KUKA KRL program: MyProgram_245().src

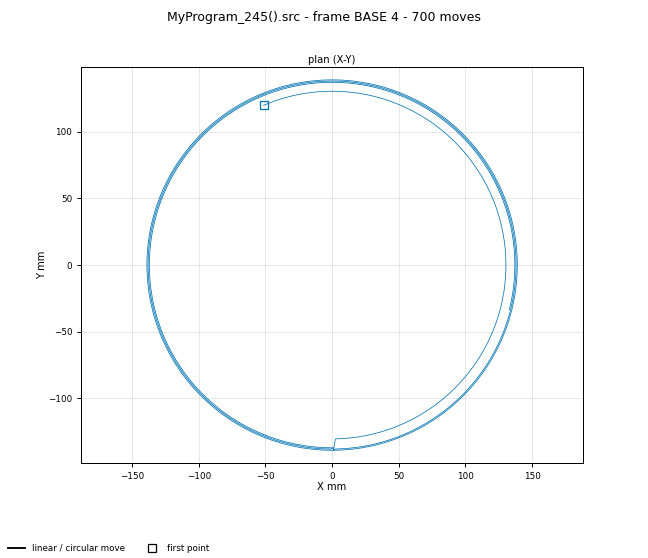
[picture p0: tool path of MyProgram_245().src in frame BASE 4, 700 of 700 moves have a stored position in this frame; points joined in program order, loops and branches not executed]
&ACCESS RVP
&REL 1
&PARAM TEMPLATE = C:\KRC\Roboter\Template\vorgabe
&PARAM EDITMASK = *
DEF MyProgram_245()
; ---- Setting reference (Base) ----
$BASE = BASE_DATA[4]

; --------------------------
; ---- Setting tool (TCP) ----
$TOOL = TOOL_DATA[3]
; --------------------------

$VEL.CP = VEL_APROX_PRINT
Startdeposition()
$VEL.CP = VEL_PRINT
LIN {X -51.3648,Y 119.8382,Z 162,A 112.229,B 13.3996,C -0.1433,E1 13.3387,E2 337.7554} C_DIS
LIN {X -48.41,Y 121.0619,Z 162,A 110.818,B 13.3996,C -0.1448,E1 13.3424,E2 339.1659} C_DIS
LIN {X -45.4271,Y 122.2124,Z 162,A 109.4036,B 13.3996,C -0.1461,E1 13.3461,E2 340.5802} C_DIS
LIN {X -41.7334,Y 123.5235,Z 162,A 107.6109,B 13.3996,C -0.1461,E1 13.3508,E2 342.3795} C_DIS
LIN {X -37.8366,Y 124.7715,Z 162,A 105.8754,B 13.3995,C -0.1495,E1 13.3554,E2 344.1065} C_DIS
LIN {X -34.901,Y 125.624,Z 162,A 104.5108,B 13.3995,C -0.1501,E1 13.3591,E2 345.4724} C_DIS
LIN {X -31.641,Y 126.4851,Z 162,A 102.9054,B 13.3995,C -0.1482,E1 13.3635,E2 347.0909} C_DIS
LIN {X -27.3855,Y 127.4735,Z 162,A 101.0691,B 13.3995,C -0.1517,E1 13.3684,E2 348.9163} C_DIS
LIN {X -23.8932,Y 128.1754,Z 162,A 99.5551,B 13.3995,C -0.154,E1 13.3726,E2 350.4234} C_DIS
LIN {X -20.7831,Y 128.7167,Z 162,A 98.1393,B 13.3995,C -0.154,E1 13.3765,E2 351.8415} C_DIS
LIN {X -17.5414,Y 129.1981,Z 162,A 96.6995,B 13.3995,C -0.1548,E1 13.3805,E2 353.2805} C_DIS
LIN {X -14.3691,Y 129.5885,Z 162,A 95.137,B 13.3995,C -0.1513,E1 13.3848,E2 354.8601} C_DIS
LIN {X -10.509,Y 129.9587,Z 162,A 93.576,B 13.3995,C -0.1556,E1 13.3891,E2 356.4038} C_DIS
LIN {X -6.3901,Y 130.2256,Z 162,A 91.7902,B 13.3995,C -0.1568,E1 13.3941,E2 358.1854} C_DIS
LIN {X -2.5144,Y 130.3584,Z 162,A 90.0176,B 13.3995,C -0.1553,E1 13.3991,E2 359.9649} C_DIS
LIN {X 0.6814,Y 130.3805,Z 162,A 88.6373,B 13.3995,C -0.156,E1 13.4029,E2 361.3419} C_DIS
LIN {X 4.7953,Y 130.2943,Z 162,A 86.8534,B 13.3995,C -0.1566,E1 13.4079,E2 363.1222} C_DIS
LIN {X 8.3824,Y 130.1129,Z 162,A 85.186,B 13.3995,C -0.1541,E1 13.4126,E2 364.7991} C_DIS
LIN {X 11.8671,Y 129.8423,Z 162,A 83.7187,B 13.3995,C -0.1557,E1 13.4166,E2 366.2581} C_DIS
LIN {X 15.283,Y 129.4833,Z 162,A 82.2394,B 13.3995,C -0.1561,E1 13.4207,E2 367.7333} C_DIS
LIN {X 18.2152,Y 129.1036,Z 162,A 80.8926,B 13.3995,C -0.1544,E1 13.4244,E2 369.0852} C_DIS
LIN {X 21.6827,Y 128.5666,Z 162,A 79.4104,B 13.3995,C -0.1554,E1 13.4285,E2 370.5601} C_DIS
LIN {X 24.8115,Y 127.9998,Z 162,A 78.0162,B 13.3995,C -0.1548,E1 13.4323,E2 371.9536} C_DIS
LIN {X 27.9273,Y 127.3565,Z 162,A 76.6207,B 13.3995,C -0.1541,E1 13.4362,E2 373.3485} C_DIS
LIN {X 31.6838,Y 126.4742,Z 162,A 74.7821,B 13.3995,C -0.1492,E1 13.4412,E2 375.2032} C_DIS
LIN {X 35.6775,Y 125.4068,Z 162,A 73.1149,B 13.3995,C -0.152,E1 13.4456,E2 376.853} C_DIS
LIN {X 39.3818,Y 124.2923,Z 162,A 71.2587,B 13.3995,C -0.1463,E1 13.4506,E2 378.727} C_DIS
LIN {X 43.2866,Y 122.988,Z 162,A 69.6267,B 13.3995,C -0.1496,E1 13.4549,E2 380.3385} C_DIS
LIN {X 46.2866,Y 121.8905,Z 162,A 68.2137,B 13.3995,C -0.148,E1 13.4586,E2 381.7524} C_DIS
LIN {X 49.8892,Y 120.4599,Z 162,A 66.4224,B 13.3995,C -0.1437,E1 13.4632,E2 383.5538} C_DIS
LIN {X 53.6946,Y 118.8129,Z 162,A 64.5724,B 13.3995,C -0.1409,E1 13.468,E2 385.4071} C_DIS
LIN {X 57.8056,Y 116.867,Z 162,A 62.6784,B 13.3995,C -0.1414,E1 13.4727,E2 387.2891} C_DIS
LIN {X 61.4635,Y 114.9879,Z 162,A 60.9224,B 13.3995,C -0.1405,E1 13.477,E2 389.0395} C_DIS
LIN {X 64.2616,Y 113.4482,Z 162,A 59.5277,B 13.3995,C -0.1388,E1 13.4804,E2 390.4334} C_DIS
LIN {X 67.0341,Y 111.8321,Z 162,A 57.9785,B 13.3997,C -0.1328,E1 13.4842,E2 391.999} C_DIS
LIN {X 70.5604,Y 109.6413,Z 162,A 56.3411,B 13.3997,C -0.1353,E1 13.488,E2 393.6151} C_DIS
LIN {X 73.2045,Y 107.8935,Z 162,A 54.9184,B 13.3997,C -0.1322,E1 13.4913,E2 395.0416} C_DIS
LIN {X 76.3807,Y 105.6688,Z 162,A 53.2322,B 13.3997,C -0.1299,E1 13.4952,E2 396.7262} C_DIS
LIN {X 79.5821,Y 103.2797,Z 162,A 51.4056,B 13.3997,C -0.1248,E1 13.4993,E2 398.5616} C_DIS
LIN {X 82.7084,Y 100.7932,Z 162,A 49.6058,B 13.3997,C -0.1204,E1 13.5032,E2 400.3672} C_DIS
LIN {X 86.1178,Y 97.8964,Z 162,A 47.6543,B 13.3997,C -0.1171,E1 13.5073,E2 402.3178} C_DIS
LIN {X 89.3226,Y 94.981,Z 162,A 45.8282,B 13.3998,C -0.1156,E1 13.511,E2 404.1357} C_DIS
LIN {X 92.196,Y 92.1952,Z 162,A 44.047,B 13.3998,C -0.1114,E1 13.5146,E2 405.9204} C_DIS
LIN {X 94.98,Y 89.3237,Z 162,A 42.3244,B 13.3998,C -0.1087,E1 13.5179,E2 407.6398} C_DIS
LIN {X 97.8953,Y 86.119,Z 162,A 40.4215,B 13.3999,C -0.1046,E1 13.5214,E2 409.5436} C_DIS
LIN {X 100.577,Y 82.9711,Z 162,A 38.6615,B 13.3999,C -0.1023,E1 13.5246,E2 411.298} C_DIS
LIN {X 103.0711,Y 79.8514,Z 162,A 36.9109,B 13.3999,C -0.0984,E1 13.5276,E2 413.0491} C_DIS
LIN {X 105.6784,Y 76.3675,Z 162,A 35.0847,B 13.3999,C -0.0964,E1 13.5306,E2 414.8666} C_DIS
LIN {X 107.8606,Y 73.2531,Z 162,A 33.3672,B 13.3999,C -0.091,E1 13.5334,E2 416.5905} C_DIS
LIN {X 109.7275,Y 70.4258,Z 162,A 31.8007,B 13.4,C -0.0851,E1 13.5358,E2 418.1672} C_DIS
LIN {X 112.0026,Y 66.748,Z 162,A 29.9637,B 13.4,C -0.0822,E1 13.5384,E2 419.9982} C_DIS
LIN {X 113.8971,Y 63.4622,Z 162,A 28.287,B 13.4,C -0.0777,E1 13.5407,E2 421.6773} C_DIS
LIN {X 116.0401,Y 59.4489,Z 162,A 26.3867,B 13.4,C -0.0754,E1 13.5432,E2 423.5676} C_DIS
LIN {X 117.5653,Y 56.3719,Z 162,A 24.978,B 13.4,C -0.0744,E1 13.5449,E2 424.9657} C_DIS
LIN {X 119.0932,Y 53.0681,Z 162,A 23.3299,B 13.4001,C -0.0687,E1 13.5468,E2 426.6209} C_DIS
LIN {X 120.4588,Y 49.8919,Z 162,A 21.8599,B 13.4001,C -0.0661,E1 13.5484,E2 428.0865} C_DIS
LIN {X 121.6461,Y 46.9227,Z 162,A 20.4706,B 13.4001,C -0.0627,E1 13.5498,E2 429.4752} C_DIS
LIN {X 122.9568,Y 43.3767,Z 162,A 18.7812,B 13.4001,C -0.0572,E1 13.5514,E2 431.1694} C_DIS
LIN {X 124.0954,Y 39.9981,Z 162,A 17.1481,B 13.4002,C -0.0509,E1 13.5529,E2 432.8117} C_DIS
LIN {X 125.2249,Y 36.308,Z 162,A 15.6024,B 13.4002,C -0.0506,E1 13.5541,E2 434.3415} C_DIS
LIN {X 126.0759,Y 33.2329,Z 162,A 14.2165,B 13.4002,C -0.0471,E1 13.5551,E2 435.7269} C_DIS
LIN {X 126.8513,Y 30.1389,Z 162,A 12.8316,B 13.4002,C -0.0435,E1 13.556,E2 437.1112} C_DIS
LIN {X 127.5503,Y 27.0298,Z 162,A 11.4491,B 13.4002,C -0.04,E1 13.5568,E2 438.4931} C_DIS
LIN {X 128.172,Y 23.9106,Z 162,A 10.0677,B 13.4002,C -0.0364,E1 13.5576,E2 439.874} C_DIS
LIN {X 128.7292,Y 20.7083,Z 162,A 8.6371,B 13.4002,C -0.0322,E1 13.5582,E2 441.3064} C_DIS
LIN {X 129.1974,Y 17.5462,Z 162,A 7.2474,B 13.4002,C -0.0285,E1 13.5588,E2 442.6959} C_DIS
LIN {X 129.588,Y 14.3743,Z 162,A 5.7046,B 13.4002,C -0.0202,E1 13.5593,E2 444.2564} C_DIS
LIN {X 129.9579,Y 10.5182,Z 162,A 4.1609,B 13.4002,C -0.0199,E1 13.5597,E2 445.7833} C_DIS
LIN {X 130.1912,Y 7.0747,Z 162,A 2.7517,B 13.4002,C -0.0187,E1 13.5599,E2 447.1816} C_DIS
LIN {X 130.3247,Y 3.8815,Z 162,A 1.1882,B 13.4002,C -0.0097,E1 13.5601,E2 448.7654} C_DIS
LIN {X 130.3848,Y 0.1344,Z 162,A -0.3942,B 13.4003,C -0.0067,E1 13.5601,E2 450.3422} C_DIS
LIN {X 130.3585,Y -2.5119,Z 162,A -1.618,B 13.4003,C -0.0014,E1 13.5601,E2 451.5745} C_DIS
LIN {X 130.2251,Y -6.3989,Z 162,A -3.2663,B 13.4003,C 0.0019,E1 13.5598,E2 453.2176} C_DIS
LIN {X 129.9591,Y -10.5042,Z 162,A -4.89,B 13.4003,C 0.0017,E1 13.5595,E2 454.8217} C_DIS
LIN {X 129.6619,Y -13.6875,Z 162,A -6.3508,B 13.4003,C 0.0076,E1 13.5591,E2 456.2907} C_DIS
LIN {X 129.2869,Y -16.8636,Z 162,A -7.6852,B 13.4003,C 0.0096,E1 13.5587,E2 457.6185} C_DIS
LIN {X 128.8327,Y -20.0401,Z 162,A -9.1175,B 13.4003,C 0.0145,E1 13.5581,E2 459.0551} C_DIS
LIN {X 128.2705,Y -23.3733,Z 162,A -10.5754,B 13.4003,C 0.018,E1 13.5574,E2 460.5116} C_DIS
LIN {X 127.6866,Y -26.3768,Z 162,A -11.922,B 13.4003,C 0.0221,E1 13.5566,E2 461.8601} C_DIS
LIN {X 127.0065,Y -29.4789,Z 162,A -13.3152,B 13.4003,C 0.0261,E1 13.5558,E2 463.2547} C_DIS
LIN {X 125.9936,Y -33.5417,Z 162,A -15.217,B 13.4003,C 0.0333,E1 13.5545,E2 465.1661} C_DIS
LIN {X 124.9621,Y -37.2055,Z 162,A -16.9347,B 13.4003,C 0.0396,E1 13.5531,E2 466.8912} C_DIS
LIN {X 123.5101,Y -41.7736,Z 162,A -18.8648,B 13.4003,C 0.0403,E1 13.5515,E2 468.8031} C_DIS
LIN {X 122.2133,Y -45.4248,Z 162,A -20.5475,B 13.4003,C 0.0445,E1 13.5499,E2 470.4855} C_DIS
LIN {X 120.7527,Y -49.1771,Z 162,A -22.324,B 13.4003,C 0.0497,E1 13.548,E2 472.2651} C_DIS
LIN {X 119.4381,Y -52.2904,Z 162,A -23.7684,B 13.4003,C 0.0526,E1 13.5464,E2 473.7065} C_DIS
LIN {X 117.86,Y -55.7553,Z 162,A -25.5751,B 13.4002,C 0.0613,E1 13.5443,E2 475.5311} C_DIS
LIN {X 116.0429,Y -59.4433,Z 162,A -27.3002,B 13.4002,C 0.0638,E1 13.5421,E2 477.2488} C_DIS
LIN {X 113.8942,Y -63.4675,Z 162,A -29.2997,B 13.4002,C 0.069,E1 13.5395,E2 479.2503} C_DIS
LIN {X 111.8352,Y -67.0289,Z 162,A -30.9899,B 13.4002,C 0.0702,E1 13.5371,E2 480.9287} C_DIS
LIN {X 109.7887,Y -70.3302,Z 162,A -32.6796,B 13.4002,C 0.0741,E1 13.5346,E2 482.6185} C_DIS
LIN {X 107.8875,Y -73.2133,Z 162,A -34.1796,B 13.4001,C 0.0775,E1 13.5323,E2 484.1183} C_DIS
LIN {X 105.67,Y -76.3791,Z 162,A -35.979,B 13.4001,C 0.0848,E1 13.5293,E2 485.9318} C_DIS
LIN {X 103.2272,Y -79.6499,Z 162,A -37.7816,B 13.4001,C 0.0894,E1 13.5263,E2 487.7375} C_DIS
LIN {X 100.5472,Y -83.0071,Z 162,A -39.5954,B 13.4,C 0.0918,E1 13.5231,E2 489.5448} C_DIS
LIN {X 97.8942,Y -86.1203,Z 162,A -41.3629,B 13.4,C 0.0951,E1 13.5199,E2 491.3109} C_DIS
LIN {X 95.1164,Y -89.1791,Z 162,A -43.2237,B 13.4,C 0.1006,E1 13.5163,E2 493.1792} C_DIS
LIN {X 92.1564,Y -92.2345,Z 162,A -45.0418,B 13.4,C 0.1032,E1 13.5128,E2 494.9933} C_DIS
LIN {X 89.3105,Y -94.9924,Z 162,A -46.7553,B 13.3999,C 0.1062,E1 13.5093,E2 496.7055} C_DIS
LIN {X 86.1673,Y -97.8526,Z 162,A -48.6377,B 13.3999,C 0.1105,E1 13.5054,E2 498.5918} C_DIS
LIN {X 82.9551,Y -100.5903,Z 162,A -50.4234,B 13.3999,C 0.1122,E1 13.5016,E2 500.3714} C_DIS
LIN {X 79.843,Y -103.0775,Z 162,A -52.1734,B 13.3999,C 0.1156,E1 13.4978,E2 502.1232} C_DIS
LIN {X 77.1216,Y -105.1292,Z 162,A -53.6275,B 13.3998,C 0.1172,E1 13.4945,E2 503.5738} C_DIS
LIN {X 73.7716,Y -107.5064,Z 162,A -55.3844,B 13.3998,C 0.1191,E1 13.4905,E2 505.3268} C_DIS
LIN {X 70.5219,Y -109.666,Z 162,A -57.1358,B 13.3998,C 0.1231,E1 13.4864,E2 507.0844} C_DIS
LIN {X 67.6092,Y -111.485,Z 162,A -58.5789,B 13.3998,C 0.1238,E1 13.483,E2 508.5212} C_DIS
LIN {X 64.8583,Y -113.1078,Z 162,A -59.9789,B 13.3998,C 0.1259,E1 13.4796,E2 509.9222} C_DIS
LIN {X 61.4575,Y -114.9911,Z 162,A -61.8495,B 13.3997,C 0.1333,E1 13.4749,E2 511.8137} C_DIS
LIN {X 57.8054,Y -116.8671,Z 162,A -63.582,B 13.3997,C 0.1339,E1 13.4706,E2 513.5393} C_DIS
LIN {X 54.3123,Y -118.5316,Z 162,A -65.1666,B 13.3997,C 0.1329,E1 13.4667,E2 515.1117} C_DIS
LIN {X 51.3578,Y -119.8413,Z 162,A -66.5759,B 13.3997,C 0.1345,E1 13.4631,E2 516.5211} C_DIS
LIN {X 48.4058,Y -121.0636,Z 162,A -67.9724,B 13.3997,C 0.136,E1 13.4594,E2 517.9179} C_DIS
LIN {X 45.4242,Y -122.2135,Z 162,A -69.3694,B 13.3997,C 0.1375,E1 13.4558,E2 519.3152} C_DIS
LIN {X 41.7737,Y -123.5101,Z 162,A -71.1872,B 13.3996,C 0.1427,E1 13.451,E2 521.1482} C_DIS
LIN {X 38.3453,Y -124.6158,Z 162,A -72.7502,B 13.3996,C 0.1437,E1 13.4468,E2 522.7101} C_DIS
LIN {X 34.7135,Y -125.6764,Z 162,A -74.2918,B 13.3996,C 0.1419,E1 13.4427,E2 524.2387} C_DIS
LIN {X 31.3975,Y -126.5469,Z 162,A -75.9774,B 13.3995,C 0.1483,E1 13.4381,E2 525.9467} C_DIS
LIN {X 26.998,Y -127.5572,Z 162,A -77.7693,B 13.3995,C 0.1444,E1 13.4332,E2 527.7173} C_DIS
LIN {X 23.9433,Y -128.1658,Z 162,A -79.1368,B 13.3995,C 0.1454,E1 13.4295,E2 529.0855} C_DIS
LIN {X 20.714,Y -128.7282,Z 162,A -80.5881,B 13.3995,C 0.1466,E1 13.4255,E2 530.5391} C_DIS
LIN {X 17.8284,Y -129.1588,Z 162,A -81.9277,B 13.3995,C 0.1489,E1 13.4218,E2 531.8863} C_DIS
LIN {X 14.3642,Y -129.5891,Z 162,A -83.5544,B 13.3995,C 0.1522,E1 13.4172,E2 533.5249} C_DIS
LIN {X 10.5051,Y -129.9591,Z 162,A -85.1137,B 13.3995,C 0.1489,E1 13.4129,E2 535.0681} C_DIS
LIN {X 6.3995,Y -130.2251,Z 162,A -86.8884,B 13.3995,C 0.1486,E1 13.408,E2 536.8399} C_DIS
LIN {X 2.5092,Y -130.3585,Z 162,A -88.632,B 13.3995,C 0.1499,E1 13.4031,E2 538.5883} C_DIS
LIN {X 2.5092,Y -130.3585,Z 162,A -88.632,B 13.3995,C 0.1499,E1 13.4031,E2 538.5883} C_DIS
Enddeposition()
LIN {X 0.9764,Y -138.8979,Z 163,A -92.574,B 24.9723,C -1.2156,E1 25.0012,E2 539.334} C_DIS
Startdeposition()
$VEL.CP = VEL_PRINT
LIN {X -2.6014,Y -138.8804,Z 163,A -94.2722,B 24.9729,C -1.203,E1 24.9963,E2 541.0621} C_DIS
LIN {X -5.7121,Y -138.7872,Z 163,A -95.5603,B 24.9729,C -1.2026,E1 24.9927,E2 542.3514} C_DIS
LIN {X -9.5587,Y -138.5762,Z 163,A -97.2235,B 24.9731,C -1.1985,E1 24.9881,E2 544.0249} C_DIS
LIN {X -13.6038,Y -138.2369,Z 163,A -98.8717,B 24.9731,C -1.2,E1 24.9835,E2 545.6702} C_DIS
LIN {X -17.9643,Y -137.7377,Z 163,A -100.6653,B 24.973,C -1.2013,E1 24.9785,E2 547.4622} C_DIS
LIN {X -21.6009,Y -137.2148,Z 163,A -102.1377,B 24.9729,C -1.204,E1 24.9745,E2 548.9293} C_DIS
LIN {X -25.0156,Y -136.6341,Z 163,A -103.5921,B 24.9729,C -1.2031,E1 24.9705,E2 550.3873} C_DIS
LIN {X -30.6353,Y -135.484,Z 163,A -105.7443,B 24.9723,C -1.2158,E1 24.9647,E2 552.5119} C_DIS
LIN {X -34.265,Y -134.6115,Z 163,A -107.5105,B 24.9728,C -1.2044,E1 24.9598,E2 554.3077} C_DIS
LIN {X -37.6332,Y -133.7091,Z 163,A -108.97,B 24.9728,C -1.2042,E1 24.9559,E2 555.7699} C_DIS
LIN {X -41.7719,Y -132.4752,Z 163,A -110.7909,B 24.9728,C -1.2034,E1 24.951,E2 557.5958} C_DIS
LIN {X -45.7264,Y -131.162,Z 163,A -112.4532,B 24.9727,C -1.2079,E1 24.9466,E2 559.2506} C_DIS
LIN {X -49.4255,Y -129.8152,Z 163,A -114.0534,B 24.9726,C -1.2107,E1 24.9424,E2 560.8475} C_DIS
LIN {X -52.632,Y -128.5486,Z 163,A -115.574,B 24.9727,C -1.2068,E1 24.9385,E2 562.3805} C_DIS
LIN {X -56.3488,Y -126.9616,Z 163,A -117.6354,B 24.9736,C -1.1877,E1 24.9331,E2 564.4921} C_DIS
LIN {X -60.2759,Y -125.145,Z 163,A -118.9432,B 24.9723,C -1.2153,E1 24.9299,E2 565.7379} C_DIS
LIN {X -63.3127,Y -123.6361,Z 163,A -120.3997,B 24.9723,C -1.214,E1 24.9263,E2 567.2014} C_DIS
LIN {X -67.2155,Y -121.5603,Z 163,A -122.2566,B 24.9723,C -1.2147,E1 24.9217,E2 569.0618} C_DIS
LIN {X -71.0183,Y -119.3786,Z 163,A -124.0755,B 24.9723,C -1.2168,E1 24.9173,E2 570.8811} C_DIS
LIN {X -74.7874,Y -117.0542,Z 163,A -125.9138,B 24.9722,C -1.2191,E1 24.913,E2 572.7199} C_DIS
LIN {X -78.5104,Y -114.5903,Z 163,A -127.7923,B 24.9722,C -1.2202,E1 24.9086,E2 574.602} C_DIS
LIN {X -82.4749,Y -111.7712,Z 163,A -129.7224,B 24.9718,C -1.2278,E1 24.9043,E2 576.5209} C_DIS
LIN {X -85.7651,Y -109.2665,Z 163,A -131.4969,B 24.9718,C -1.2273,E1 24.9003,E2 578.3029} C_DIS
LIN {X -89.2892,Y -106.4061,Z 163,A -133.3216,B 24.9715,C -1.2334,E1 24.8964,E2 580.12} C_DIS
LIN {X -92.8718,Y -103.2943,Z 163,A -135.244,B 24.9712,C -1.2392,E1 24.8924,E2 582.0363} C_DIS
LIN {X -95.8142,Y -100.5709,Z 163,A -137.0274,B 24.9714,C -1.2359,E1 24.8887,E2 583.8348} C_DIS
LIN {X -99.0965,Y -97.3381,Z 163,A -138.8571,B 24.971,C -1.2438,E1 24.8851,E2 585.6535} C_DIS
LIN {X -102.0916,Y -94.1923,Z 163,A -141.3701,B 24.9726,C -1.2105,E1 24.8802,E2 588.2566} C_DIS
LIN {X -105.9427,Y -89.8388,Z 163,A -143.0142,B 24.9705,C -1.2551,E1 24.8774,E2 589.8021} C_DIS
LIN {X -108.4906,Y -86.7451,Z 163,A -144.8147,B 24.9707,C -1.2515,E1 24.8742,E2 591.6196} C_DIS
LIN {X -111.357,Y -83.0328,Z 163,A -146.5333,B 24.9699,C -1.2676,E1 24.8713,E2 593.3082} C_DIS
LIN {X -113.2795,Y -80.3911,Z 163,A -148.1107,B 24.9703,C -1.2591,E1 24.8687,E2 594.9134} C_DIS
LIN {X -116.4336,Y -75.75,Z 163,A -150.416,B 24.97,C -1.2657,E1 24.8651,E2 597.2145} C_DIS
LIN {X -118.8488,Y -71.9013,Z 163,A -152.3177,B 24.9698,C -1.2694,E1 24.8623,E2 599.1172} C_DIS
LIN {X -121.2689,Y -67.7409,Z 163,A -154.2352,B 24.9694,C -1.2784,E1 24.8597,E2 601.0233} C_DIS
LIN {X -123.3829,Y -63.8097,Z 163,A -156.0537,B 24.9691,C -1.2847,E1 24.8573,E2 602.8363} C_DIS
LIN {X -124.8311,Y -60.9246,Z 163,A -157.3948,B 24.9689,C -1.2881,E1 24.8557,E2 604.1766} C_DIS
LIN {X -126.9365,Y -56.4049,Z 163,A -159.4973,B 24.9687,C -1.2918,E1 24.8532,E2 606.2818} C_DIS
LIN {X -128.3923,Y -53.0097,Z 163,A -161.1335,B 24.9688,C -1.2906,E1 24.8514,E2 607.93} C_DIS
LIN {X -130.3375,Y -48.031,Z 163,A -163.1898,B 24.9681,C -1.3048,E1 24.8494,E2 609.964} C_DIS
LIN {X -131.3369,Y -45.2217,Z 163,A -164.4694,B 24.9681,C -1.3061,E1 24.8482,E2 611.2479} C_DIS
LIN {X -133.1593,Y -39.5374,Z 163,A -167.0872,B 24.9681,C -1.3058,E1 24.846,E2 613.8815} C_DIS
LIN {X -134.4482,Y -34.9084,Z 163,A -169.0525,B 24.9677,C -1.3128,E1 24.8446,E2 615.8413} C_DIS
LIN {X -135.439,Y -30.8323,Z 163,A -170.6194,B 24.967,C -1.3267,E1 24.8436,E2 617.3843} C_DIS
LIN {X -136.0751,Y -27.892,Z 163,A -171.9327,B 24.967,C -1.327,E1 24.8429,E2 618.7046} C_DIS
LIN {X -136.7453,Y -24.3947,Z 163,A -173.3649,B 24.9667,C -1.3336,E1 24.8421,E2 620.1296} C_DIS
LIN {X -137.2596,Y -21.3116,Z 163,A -174.654,B 24.9665,C -1.3378,E1 24.8416,E2 621.4165} C_DIS
LIN {X -137.726,Y -18.0534,Z 163,A -176.0597,B 24.9664,C -1.3398,E1 24.841,E2 622.8258} C_DIS
LIN {X -138.1515,Y -14.4475,Z 163,A -177.5509,B 24.9661,C -1.345,E1 24.8406,E2 624.3134} C_DIS
LIN {X -138.4495,Y -11.24,Z 163,A -178.8872,B 24.9659,C -1.349,E1 24.8402,E2 625.6483} C_DIS
LIN {X -138.6778,Y -7.9514,Z 163,A 179.7547,B 24.9657,C -1.3535,E1 24.84,E2 627.0037} C_DIS
LIN {X -138.8293,Y -4.6292,Z 163,A 178.2111,B 24.9659,C -1.3494,E1 24.8398,E2 628.5666} C_DIS
LIN {X -138.9061,Y -0.3225,Z 163,A 176.1204,B 24.9664,C -1.3394,E1 24.8398,E2 630.6935} C_DIS
LIN {X -138.8572,Y 3.628,Z 163,A 175.1219,B 24.9645,C -1.3768,E1 24.8398,E2 631.6091} C_DIS
LIN {X -138.7897,Y 5.6476,Z 163,A 173.7018,B 24.9659,C -1.3499,E1 24.84,E2 633.1019} C_DIS
LIN {X -138.5822,Y 9.4763,Z 163,A 172.3725,B 24.965,C -1.3678,E1 24.8403,E2 634.3963} C_DIS
LIN {X -138.2645,Y 13.316,Z 163,A 170.9058,B 24.9644,C -1.3793,E1 24.8406,E2 635.8444} C_DIS
LIN {X -137.9208,Y 16.4998,Z 163,A 169.5737,B 24.9642,C -1.3831,E1 24.841,E2 637.1754} C_DIS
LIN {X -137.506,Y 19.6594,Z 163,A 168.2372,B 24.964,C -1.3864,E1 24.8415,E2 638.5121} C_DIS
LIN {X -136.988,Y 22.9931,Z 163,A 166.8391,B 24.9638,C -1.3907,E1 24.8422,E2 639.9084} C_DIS
LIN {X -136.3581,Y 26.4763,Z 163,A 165.3401,B 24.9636,C -1.3935,E1 24.8429,E2 641.4094} C_DIS
LIN {X -135.6047,Y 30.1057,Z 163,A 163.6793,B 24.9637,C -1.3918,E1 24.8439,E2 643.084} C_DIS
LIN {X -134.6219,Y 34.224,Z 163,A 162.106,B 24.963,C -1.4064,E1 24.8449,E2 644.6319} C_DIS
LIN {X -133.815,Y 37.2545,Z 163,A 160.6974,B 24.963,C -1.4048,E1 24.846,E2 646.0526} C_DIS
LIN {X -132.8233,Y 40.6484,Z 163,A 159.3287,B 24.9625,C -1.414,E1 24.8471,E2 647.407} C_DIS
LIN {X -131.3327,Y 45.234,Z 163,A 157.4975,B 24.9618,C -1.4284,E1 24.8487,E2 649.2144} C_DIS
LIN {X -128.5676,Y 52.5849,Z 163,A 154.0243,B 24.9618,C -1.4267,E1 24.8522,E2 652.7112} C_DIS
LIN {X -127.3209,Y 55.5325,Z 163,A 152.6939,B 24.9617,C -1.4304,E1 24.8536,E2 654.0403} C_DIS
LIN {X -125.7517,Y 59.0032,Z 163,A 151.0079,B 24.9617,C -1.4294,E1 24.8556,E2 655.7379} C_DIS
LIN {X -123.9243,Y 62.7465,Z 163,A 149.3216,B 24.9614,C -1.4363,E1 24.8577,E2 657.4168} C_DIS
LIN {X -122.0533,Y 66.3164,Z 163,A 147.4756,B 24.9616,C -1.432,E1 24.8601,E2 659.2829} C_DIS
LIN {X -120.0216,Y 69.9271,Z 163,A 145.298,B 24.9626,C -1.4134,E1 24.8633,E2 661.516} C_DIS
LIN {X -117.1735,Y 74.601,Z 163,A 143.3303,B 24.9614,C -1.4346,E1 24.8661,E2 663.4432} C_DIS
LIN {X -115.0883,Y 77.7787,Z 163,A 142.0457,B 24.9604,C -1.4534,E1 24.8681,E2 664.6893} C_DIS
LIN {X -112.2037,Y 81.8858,Z 163,A 139.9914,B 24.9601,C -1.4601,E1 24.8714,E2 666.7379} C_DIS
LIN {X -109.7279,Y 85.1741,Z 163,A 138.2918,B 24.9598,C -1.4647,E1 24.8743,E2 668.4346} C_DIS
LIN {X -107.2853,Y 88.2315,Z 163,A 136.7189,B 24.9595,C -1.4711,E1 24.877,E2 669.9994} C_DIS
LIN {X -105.1466,Y 90.7691,Z 163,A 135.262,B 24.9595,C -1.4703,E1 24.8797,E2 671.465} C_DIS
LIN {X -102.1717,Y 94.1051,Z 163,A 133.4056,B 24.9593,C -1.4744,E1 24.8832,E2 673.3199} C_DIS
LIN {X -99.069,Y 97.3662,Z 163,A 131.5746,B 24.9589,C -1.4804,E1 24.8867,E2 675.1445} C_DIS
LIN {X -95.8896,Y 100.4989,Z 163,A 129.6866,B 24.9589,C -1.4825,E1 24.8905,E2 677.0352} C_DIS
LIN {X -92.5636,Y 103.5704,Z 163,A 127.8048,B 24.9586,C -1.4862,E1 24.8944,E2 678.9158} C_DIS
LIN {X -89.1155,Y 106.5519,Z 163,A 125.9386,B 24.9583,C -1.4913,E1 24.8983,E2 680.7772} C_DIS
LIN {X -85.5843,Y 109.4085,Z 163,A 124.052,B 24.9581,C -1.4948,E1 24.9024,E2 682.6626} C_DIS
LIN {X -82.1675,Y 111.9971,Z 163,A 122.2902,B 24.9579,C -1.4989,E1 24.9064,E2 684.4208} C_DIS
LIN {X -78.6359,Y 114.5042,Z 163,A 120.4821,B 24.9578,C -1.5015,E1 24.9105,E2 686.229} C_DIS
LIN {X -75.3596,Y 116.6871,Z 163,A 118.7994,B 24.9578,C -1.5017,E1 24.9145,E2 687.9168} C_DIS
LIN {X -72.1263,Y 118.7127,Z 163,A 117.2266,B 24.9576,C -1.5047,E1 24.9182,E2 689.4872} C_DIS
LIN {X -68.2663,Y 120.9735,Z 163,A 115.4147,B 24.9573,C -1.5098,E1 24.9226,E2 691.2924} C_DIS
LIN {X -62.8152,Y 123.8894,Z 163,A 112.9208,B 24.9569,C -1.5171,E1 24.9287,E2 693.7757} C_DIS
LIN {X -59.4989,Y 125.5163,Z 163,A 111.3272,B 24.9569,C -1.516,E1 24.9327,E2 695.3763} C_DIS
LIN {X -54.735,Y 127.6658,Z 163,A 109.3096,B 24.9563,C -1.5265,E1 24.9378,E2 697.3738} C_DIS
LIN {X -48.1619,Y 130.2885,Z 163,A 106.3577,B 24.9563,C -1.5288,E1 24.9455,E2 700.3265} C_DIS
LIN {X -45.2605,Y 131.3235,Z 163,A 105.1243,B 24.956,C -1.5324,E1 24.9487,E2 701.5537} C_DIS
LIN {X -42.2172,Y 132.333,Z 163,A 103.6746,B 24.9563,C -1.5273,E1 24.9526,E2 703.0183} C_DIS
LIN {X -37.1719,Y 133.8381,Z 163,A 101.565,B 24.956,C -1.533,E1 24.9583,E2 705.1177} C_DIS
LIN {X -33.9118,Y 134.7012,Z 163,A 100.1128,B 24.956,C -1.5312,E1 24.9622,E2 706.5764} C_DIS
LIN {X -30.2855,Y 135.5639,Z 163,A 98.6212,B 24.9559,C -1.535,E1 24.9662,E2 708.0608} C_DIS
LIN {X -27.1782,Y 136.2203,Z 163,A 97.3241,B 24.9557,C -1.5369,E1 24.9698,E2 709.3551} C_DIS
LIN {X -23.7281,Y 136.8646,Z 163,A 95.5116,B 24.9568,C -1.5186,E1 24.9749,E2 711.2127} C_DIS
LIN {X -20.3572,Y 137.4049,Z 163,A 94.358,B 24.956,C -1.5331,E1 24.978,E2 712.3329} C_DIS
LIN {X -16.4641,Y 137.9251,Z 163,A 92.3738,B 24.957,C -1.5148,E1 24.9836,E2 714.362} C_DIS
LIN {X -12.2896,Y 138.3609,Z 163,A 91.1729,B 24.9553,C -1.5439,E1 24.9868,E2 715.4945} C_DIS
LIN {X -9.7251,Y 138.564,Z 163,A 89.9539,B 24.9558,C -1.5359,E1 24.9902,E2 716.733} C_DIS
LIN {X -5.4451,Y 138.7976,Z 163,A 88.2248,B 24.9556,C -1.5386,E1 24.995,E2 718.4561} C_DIS
LIN {X -0.8368,Y 138.9019,Z 163,A 86.1925,B 24.956,C -1.532,E1 25.0007,E2 720.504} C_DIS
LIN {X 3.7428,Y 138.854,Z 163,A 84.4393,B 24.9556,C -1.5396,E1 25.0056,E2 722.239} C_DIS
LIN {X 7.8483,Y 138.6842,Z 163,A 82.6991,B 24.9557,C -1.5372,E1 25.0104,E2 723.9843} C_DIS
LIN {X 12.3027,Y 138.3597,Z 163,A 80.6656,B 24.9563,C -1.5268,E1 25.0162,E2 726.0415} C_DIS
LIN {X 16.0621,Y 137.973,Z 163,A 79.3101,B 24.9557,C -1.5375,E1 25.0198,E2 727.3706} C_DIS
LIN {X 19.7043,Y 137.4995,Z 163,A 77.7925,B 24.9557,C -1.537,E1 25.024,E2 728.8881} C_DIS
LIN {X 27.2071,Y 136.2145,Z 163,A 74.8385,B 24.9552,C -1.5458,E1 25.0321,E2 731.818} C_DIS
LIN {X 31.6736,Y 135.2468,Z 163,A 72.8351,B 24.9557,C -1.5383,E1 25.0376,E2 733.8364} C_DIS
LIN {X 34.7502,Y 134.4884,Z 163,A 71.3839,B 24.9562,C -1.5297,E1 25.0416,E2 735.306} C_DIS
LIN {X 38.9005,Y 133.3458,Z 163,A 69.6919,B 24.956,C -1.533,E1 25.0461,E2 736.9873} C_DIS
LIN {X 42.5914,Y 132.2135,Z 163,A 68.1573,B 24.9559,C -1.5349,E1 25.0502,E2 738.5146} C_DIS
LIN {X 46.1437,Y 131.0173,Z 163,A 66.5424,B 24.9562,C -1.5297,E1 25.0545,E2 740.1386} C_DIS
LIN {X 50.0604,Y 129.5698,Z 163,A 64.8155,B 24.9562,C -1.5278,E1 25.059,E2 741.8664} C_DIS
LIN {X 54.3535,Y 127.8307,Z 163,A 62.6138,B 24.9573,C -1.5096,E1 25.0647,E2 744.1058} C_DIS
LIN {X 57.7236,Y 126.3435,Z 163,A 61.5539,B 24.956,C -1.5332,E1 25.0673,E2 745.1074} C_DIS
LIN {X 62.0858,Y 124.2583,Z 163,A 59.368,B 24.9567,C -1.52,E1 25.0728,E2 747.3187} C_DIS
LIN {X 66.0765,Y 122.1838,Z 163,A 57.5256,B 24.9568,C -1.5181,E1 25.0774,E2 749.1603} C_DIS
LIN {X 69.9969,Y 119.981,Z 163,A 55.6693,B 24.957,C -1.5153,E1 25.0819,E2 751.0176} C_DIS
LIN {X 73.9074,Y 117.612,Z 163,A 53.8453,B 24.957,C -1.5158,E1 25.0862,E2 752.8347} C_DIS
LIN {X 77.4526,Y 115.3086,Z 163,A 52.0469,B 24.9573,C -1.5099,E1 25.0904,E2 754.6412} C_DIS
LIN {X 81.0522,Y 112.8072,Z 163,A 50.3024,B 24.9573,C -1.5102,E1 25.0944,E2 756.3788} C_DIS
LIN {X 84.3504,Y 110.3623,Z 163,A 48.619,B 24.9574,C -1.5077,E1 25.0981,E2 758.0621} C_DIS
LIN {X 87.6177,Y 107.7873,Z 163,A 46.8802,B 24.9577,C -1.5031,E1 25.1019,E2 759.8052} C_DIS
LIN {X 90.7909,Y 105.1278,Z 163,A 45.4078,B 24.9571,C -1.513,E1 25.105,E2 761.2486} C_DIS
LIN {X 93.2782,Y 102.9272,Z 163,A 43.7897,B 24.9581,C -1.4961,E1 25.1084,E2 762.9} C_DIS
LIN {X 96.9706,Y 99.4569,Z 163,A 41.9305,B 24.9576,C -1.5047,E1 25.1122,E2 764.7313} C_DIS
LIN {X 99.1933,Y 97.2394,Z 163,A 40.473,B 24.9583,C -1.4926,E1 25.1151,E2 766.2111} C_DIS
LIN {X 104.1956,Y 91.8593,Z 163,A 37.6526,B 24.958,C -1.4975,E1 25.1204,E2 769.0075} C_DIS
LIN {X 106.4517,Y 89.2349,Z 163,A 36.0074,B 24.9589,C -1.4817,E1 25.1234,E2 770.6826} C_DIS
LIN {X 109.18,Y 85.8752,Z 163,A 34.2671,B 24.9589,C -1.4798,E1 25.1264,E2 772.4191} C_DIS
LIN {X 111.6464,Y 82.644,Z 163,A 32.587,B 24.9592,C -1.4754,E1 25.1292,E2 774.1017} C_DIS
LIN {X 114.0529,Y 79.2891,Z 163,A 30.8629,B 24.9595,C -1.4698,E1 25.132,E2 775.8307} C_DIS
LIN {X 116.5502,Y 75.5704,Z 163,A 29.0359,B 24.9597,C -1.466,E1 25.1348,E2 777.6574} C_DIS
LIN {X 118.9434,Y 71.7448,Z 163,A 27.1794,B 24.96,C -1.4612,E1 25.1375,E2 779.5158} C_DIS
LIN {X 121.1898,Y 67.8815,Z 163,A 25.347,B 24.9602,C -1.4567,E1 25.1401,E2 781.3493} C_DIS
LIN {X 123.3053,Y 63.9574,Z 163,A 23.6369,B 24.9602,C -1.4589,E1 25.1423,E2 783.0452} C_DIS
LIN {X 124.6589,Y 61.2737,Z 163,A 22.367,B 24.9604,C -1.4536,E1 25.1439,E2 784.3209} C_DIS
LIN {X 126.1684,Y 58.1021,Z 163,A 20.9235,B 24.9606,C -1.4497,E1 25.1456,E2 785.7659} C_DIS
LIN {X 127.6265,Y 54.8257,Z 163,A 19.361,B 24.9611,C -1.4405,E1 25.1474,E2 787.3414} C_DIS
LIN {X 129.347,Y 50.6337,Z 163,A 17.541,B 24.9613,C -1.4377,E1 25.1493,E2 789.1579} C_DIS
LIN {X 130.7863,Y 46.7905,Z 163,A 15.8979,B 24.9614,C -1.4354,E1 25.1508,E2 790.7973} C_DIS
LIN {X 132.1358,Y 42.8346,Z 163,A 14.0041,B 24.9622,C -1.4203,E1 25.1525,E2 792.716} C_DIS
LIN {X 133.5069,Y 38.35,Z 163,A 12.1595,B 24.9622,C -1.4194,E1 25.154,E2 794.5522} C_DIS
LIN {X 134.5985,Y 34.3162,Z 163,A 10.5143,B 24.9623,C -1.4185,E1 25.1551,E2 796.1901} C_DIS
LIN {X 135.4657,Y 30.7153,Z 163,A 9.0458,B 24.9623,C -1.417,E1 25.1561,E2 797.6535} C_DIS
LIN {X 136.2491,Y 27.0369,Z 163,A 7.4323,B 24.9628,C -1.4084,E1 25.157,E2 799.2779} C_DIS
LIN {X 137.3129,Y 20.9672,Z 163,A 5.074,B 24.9628,C -1.4108,E1 25.1581,E2 801.6167} C_DIS
LIN {X 137.7337,Y 17.9949,Z 163,A 3.7698,B 24.9631,C -1.4029,E1 25.1586,E2 802.9318} C_DIS
LIN {X 138.1641,Y 14.3309,Z 163,A 2.1917,B 24.9636,C -1.3946,E1 25.1591,E2 804.52} C_DIS
LIN {X 138.6236,Y 8.8312,Z 163,A -0.1695,B 24.9642,C -1.3822,E1 25.1596,E2 806.8965} C_DIS
LIN {X 138.8343,Y 4.4513,Z 163,A -1.912,B 24.9643,C -1.38,E1 25.1597,E2 808.6338} C_DIS
LIN {X 138.908,Y -0.012,Z 163,A -3.7222,B 24.9646,C -1.3757,E1 25.1597,E2 810.4435} C_DIS
LIN {X 138.8188,Y -4.9011,Z 163,A -5.8665,B 24.9653,C -1.3616,E1 25.1597,E2 812.6082} C_DIS
LIN {X 138.531,Y -10.1766,Z 163,A -7.8565,B 24.9651,C -1.3653,E1 25.1593,E2 814.5775} C_DIS
LIN {X 138.1104,Y -14.8297,Z 163,A -9.7403,B 24.9653,C -1.3614,E1 25.1588,E2 816.4595} C_DIS
LIN {X 137.6716,Y -18.469,Z 163,A -11.3456,B 24.9658,C -1.3509,E1 25.1582,E2 818.0799} C_DIS
LIN {X 137.1245,Y -22.1749,Z 163,A -12.704,B 24.9655,C -1.3567,E1 25.1576,E2 819.4169} C_DIS
LIN {X 136.0062,Y -28.2306,Z 163,A -15.2383,B 24.9659,C -1.3486,E1 25.1563,E2 821.9554} C_DIS
LIN {X 134.5899,Y -34.3501,Z 163,A -17.838,B 24.9664,C -1.3395,E1 25.1546,E2 824.5614} C_DIS
LIN {X 133.706,Y -37.6443,Z 163,A -19.2509,B 24.9666,C -1.3346,E1 25.1536,E2 825.9778} C_DIS
LIN {X 132.7867,Y -40.768,Z 163,A -20.5164,B 24.9666,C -1.3347,E1 25.1526,E2 827.2358} C_DIS
LIN {X 131.7174,Y -44.101,Z 163,A -21.954,B 24.9668,C -1.3304,E1 25.1513,E2 828.6754} C_DIS
LIN {X 130.5756,Y -47.3752,Z 163,A -23.4664,B 24.9673,C -1.321,E1 25.1499,E2 830.2013} C_DIS
LIN {X 129.1385,Y -51.1685,Z 163,A -25.1484,B 24.9676,C -1.3151,E1 25.1482,E2 831.8879} C_DIS
LIN {X 127.6639,Y -54.7392,Z 163,A -26.898,B 24.9683,C -1.3011,E1 25.1463,E2 833.6609} C_DIS
LIN {X 125.9702,Y -58.5309,Z 163,A -28.3918,B 24.9679,C -1.3085,E1 25.1446,E2 835.1294} C_DIS
LIN {X 124.2406,Y -62.1218,Z 163,A -30.012,B 24.9681,C -1.3047,E1 25.1426,E2 836.7496} C_DIS
LIN {X 122.5152,Y -65.4595,Z 163,A -31.6237,B 24.9685,C -1.2964,E1 25.1405,E2 838.3725} C_DIS
LIN {X 120.5132,Y -69.0759,Z 163,A -33.3003,B 24.9687,C -1.2929,E1 25.1382,E2 840.0486} C_DIS
LIN {X 118.424,Y -72.5988,Z 163,A -34.9822,B 24.9689,C -1.2883,E1 25.1357,E2 841.7327} C_DIS
LIN {X 116.284,Y -75.9804,Z 163,A -36.5995,B 24.9691,C -1.2854,E1 25.1333,E2 843.3487} C_DIS
LIN {X 114.2901,Y -78.948,Z 163,A -37.9061,B 24.9688,C -1.2909,E1 25.1313,E2 844.6359} C_DIS
LIN {X 112.4731,Y -81.5145,Z 163,A -39.4125,B 24.9695,C -1.2751,E1 25.1288,E2 846.1722} C_DIS
LIN {X 109.6912,Y -85.2214,Z 163,A -41.3362,B 24.9698,C -1.2691,E1 25.1255,E2 848.101} C_DIS
LIN {X 106.9304,Y -88.6607,Z 163,A -43.1086,B 24.9699,C -1.2668,E1 25.1224,E2 849.8705} C_DIS
LIN {X 104.0824,Y -91.9873,Z 163,A -44.94,B 24.9702,C -1.2606,E1 25.119,E2 851.7084} C_DIS
LIN {X 100.8882,Y -95.4801,Z 163,A -46.8453,B 24.9704,C -1.2582,E1 25.1154,E2 853.6109} C_DIS
LIN {X 97.9234,Y -98.5182,Z 163,A -48.5991,B 24.9706,C -1.2536,E1 25.112,E2 855.368} C_DIS
LIN {X 94.6917,Y -101.6283,Z 163,A -50.4636,B 24.9708,C -1.2483,E1 25.1082,E2 857.2375} C_DIS
LIN {X 91.5875,Y -104.435,Z 163,A -52.1925,B 24.971,C -1.244,E1 25.1045,E2 858.9697} C_DIS
LIN {X 88.0125,Y -107.4646,Z 163,A -54.0938,B 24.9711,C -1.2413,E1 25.1005,E2 860.8699} C_DIS
LIN {X 84.3697,Y -110.3475,Z 163,A -56.0009,B 24.9713,C -1.2376,E1 25.0963,E2 862.7788} C_DIS
LIN {X 81.0865,Y -112.7826,Z 163,A -57.6661,B 24.9714,C -1.2352,E1 25.0925,E2 864.4438} C_DIS
LIN {X 77.379,Y -115.3577,Z 163,A -59.5222,B 24.9716,C -1.2316,E1 25.0882,E2 866.302} C_DIS
LIN {X 73.6606,Y -117.7669,Z 163,A -61.3346,B 24.9717,C -1.2289,E1 25.084,E2 868.1151} C_DIS
LIN {X 70.0092,Y -119.9737,Z 163,A -63.0895,B 24.9719,C -1.2258,E1 25.0797,E2 869.8718} C_DIS
LIN {X 66.287,Y -122.0694,Z 163,A -64.9089,B 24.9722,C -1.2194,E1 25.0753,E2 871.7011} C_DIS
LIN {X 62.5802,Y -124.009,Z 163,A -66.4978,B 24.9719,C -1.2242,E1 25.0714,E2 873.2743} C_DIS
LIN {X 58.6985,Y -125.8926,Z 163,A -68.3264,B 24.9722,C -1.2185,E1 25.0667,E2 875.1116} C_DIS
LIN {X 51.2119,Y -129.121,Z 163,A -71.5444,B 24.9721,C -1.2215,E1 25.0585,E2 878.3148} C_DIS
LIN {X 46.4415,Y -130.9122,Z 163,A -73.6895,B 24.9723,C -1.2162,E1 25.0529,E2 880.468} C_DIS
LIN {X 43.4965,Y -131.9187,Z 163,A -75.0016,B 24.9724,C -1.213,E1 25.0494,E2 881.7852} C_DIS
LIN {X 40.1627,Y -132.9719,Z 163,A -76.3961,B 24.9724,C -1.2139,E1 25.0457,E2 883.1749} C_DIS
LIN {X 37.1179,Y -133.8532,Z 163,A -77.727,B 24.9725,C -1.2111,E1 25.0421,E2 884.5101} C_DIS
LIN {X 33.0762,Y -134.9096,Z 163,A -79.4991,B 24.9727,C -1.2065,E1 25.0373,E2 886.2904} C_DIS
LIN {X 29.2238,Y -135.7952,Z 163,A -81.4296,B 24.9736,C -1.1883,E1 25.0319,E2 888.2615} C_DIS
LIN {X 25.5151,Y -136.5418,Z 163,A -82.5962,B 24.9726,C -1.2089,E1 25.0288,E2 889.3781} C_DIS
LIN {X 22.5096,Y -137.0686,Z 163,A -83.8626,B 24.9726,C -1.2075,E1 25.0253,E2 890.6465} C_DIS
LIN {X 19.2858,Y -137.5593,Z 163,A -85.1817,B 24.9726,C -1.2079,E1 25.0217,E2 891.9633} C_DIS
LIN {X 15.783,Y -138.0063,Z 163,A -87.1049,B 24.9739,C -1.1812,E1 25.0162,E2 893.9484} C_DIS
LIN {X 11.8663,Y -138.3966,Z 163,A -88.3652,B 24.973,C -1.2004,E1 25.0128,E2 895.1625} C_DIS
LIN {X 7.8159,Y -138.6861,Z 163,A -90.0513,B 24.973,C -1.199,E1 25.0081,E2 896.8511} C_DIS
LIN {X 3.8549,Y -138.8509,Z 163,A -91.6475,B 24.973,C -1.2006,E1 25.0037,E2 898.4431} C_DIS
LIN {X 0.9764,Y -138.8979,Z 163,A -92.5722,B 24.9724,C -1.2149,E1 25.0012,E2 899.334} C_DIS
Enddeposition()
LIN {X 0.9764,Y -138.8979,Z 163,A -92.5722,B 24.9724,C -1.2149,E1 25.0012,E2 899.334} C_DIS
Startdeposition()
$VEL.CP = VEL_PRINT
LIN {X 2.2698,Y -137.9648,Z 163,A -91.6339,B 24.9706,C -1.2533,E1 25.0041,E2 898.3048} C_DIS
LIN {X 6.4017,Y -137.8359,Z 163,A -89.9534,B 24.9706,C -1.2519,E1 25.0087,E2 896.628} C_DIS
LIN {X 9.2489,Y -137.6752,Z 163,A -88.2711,B 24.9693,C -1.2802,E1 25.0136,E2 894.8794} C_DIS
LIN {X 13.5372,Y -137.3182,Z 163,A -86.9746,B 24.9706,C -1.2538,E1 25.017,E2 893.6463} C_DIS
LIN {X 20.4324,Y -136.4638,Z 163,A -84.1598,B 24.9706,C -1.2517,E1 25.0248,E2 890.8388} C_DIS
LIN {X 23.212,Y -136.0178,Z 163,A -82.3051,B 24.9688,C -1.2912,E1 25.0302,E2 888.8925} C_DIS
LIN {X 28.3291,Y -135.0462,Z 163,A -80.6572,B 24.9701,C -1.264,E1 25.0345,E2 887.311} C_DIS
LIN {X 32.1515,Y -134.1852,Z 163,A -79.1598,B 24.9703,C -1.2584,E1 25.0385,E2 885.829} C_DIS
LIN {X 35.4734,Y -133.3454,Z 163,A -77.7444,B 24.9703,C -1.2595,E1 25.0423,E2 884.4132} C_DIS
LIN {X 38.84,Y -132.4039,Z 163,A -76.2726,B 24.9702,C -1.2623,E1 25.0463,E2 882.9372} C_DIS
LIN {X 42.3683,Y -131.318,Z 163,A -74.6889,B 24.9699,C -1.267,E1 25.0505,E2 881.3453} C_DIS
LIN {X 45.9436,Y -130.112,Z 163,A -72.6502,B 24.9685,C -1.2959,E1 25.0561,E2 879.2424} C_DIS
LIN {X 50.1948,Y -128.5295,Z 163,A -71.411,B 24.9702,C -1.2619,E1 25.0591,E2 878.0862} C_DIS
LIN {X 54.1417,Y -126.9179,Z 163,A -69.3338,B 24.9692,C -1.282,E1 25.0646,E2 875.9665} C_DIS
LIN {X 59.0081,Y -124.7301,Z 163,A -67.0302,B 24.9688,C -1.2906,E1 25.0704,E2 873.6484} C_DIS
LIN {X 62.0813,Y -123.2296,Z 163,A -65.8495,B 24.9693,C -1.2793,E1 25.0733,E2 872.4976} C_DIS
LIN {X 65.4387,Y -121.481,Z 163,A -64.2841,B 24.9693,C -1.2817,E1 25.0772,E2 870.931} C_DIS
LIN {X 69.1516,Y -119.4064,Z 163,A -62.5448,B 24.9692,C -1.2834,E1 25.0814,E2 869.1927} C_DIS
LIN {X 72.7204,Y -117.2673,Z 163,A -60.7772,B 24.9689,C -1.289,E1 25.0856,E2 867.4173} C_DIS
LIN {X 76.4715,Y -114.8563,Z 163,A -58.9521,B 24.9688,C -1.2912,E1 25.0899,E2 865.593} C_DIS
LIN {X 79.8826,Y -112.5113,Z 163,A -57.1982,B 24.9685,C -1.2968,E1 25.0939,E2 863.832} C_DIS
LIN {X 83.607,Y -109.7714,Z 163,A -55.2905,B 24.9683,C -1.3003,E1 25.0982,E2 861.9228} C_DIS
LIN {X 87.2493,Y -106.899,Z 163,A -53.4347,B 24.9683,C -1.3006,E1 25.1022,E2 860.0734} C_DIS
LIN {X 90.4833,Y -104.1763,Z 163,A -51.6322,B 24.968,C -1.3075,E1 25.106,E2 858.2618} C_DIS
LIN {X 93.8816,Y -101.1243,Z 163,A -49.748,B 24.9678,C -1.3113,E1 25.1099,E2 856.3761} C_DIS
LIN {X 97.2281,Y -97.9108,Z 163,A -47.8858,B 24.9678,C -1.3124,E1 25.1136,E2 854.5191} C_DIS
LIN {X 100.186,Y -94.8823,Z 163,A -46.0785,B 24.9674,C -1.3198,E1 25.1171,E2 852.7023} C_DIS
LIN {X 103.3168,Y -91.463,Z 163,A -44.1862,B 24.9672,C -1.3229,E1 25.1207,E2 850.811} C_DIS
LIN {X 106.2872,Y -87.9935,Z 163,A -42.3015,B 24.967,C -1.3274,E1 25.1241,E2 848.9244} C_DIS
LIN {X 109.0837,Y -84.502,Z 163,A -40.5056,B 24.967,C -1.3289,E1 25.1272,E2 847.1333} C_DIS
LIN {X 111.5037,Y -81.2829,Z 163,A -38.7645,B 24.9665,C -1.3376,E1 25.1301,E2 845.3801} C_DIS
LIN {X 113.2816,Y -78.7852,Z 163,A -37.3081,B 24.9658,C -1.3519,E1 25.1325,E2 843.897} C_DIS
LIN {X 115.2009,Y -75.9512,Z 163,A -36.0519,B 24.966,C -1.3464,E1 25.1344,E2 842.6601} C_DIS
LIN {X 117.8413,Y -71.7875,Z 163,A -34.1119,B 24.966,C -1.3462,E1 25.1372,E2 840.7304} C_DIS
LIN {X 120.0161,Y -68.0887,Z 163,A -32.3711,B 24.966,C -1.3491,E1 25.1396,E2 838.9916} C_DIS
LIN {X 121.9044,Y -64.6444,Z 163,A -30.8891,B 24.966,C -1.3454,E1 25.1416,E2 837.5261} C_DIS
LIN {X 123.507,Y -61.5271,Z 163,A -29.3135,B 24.9655,C -1.3569,E1 25.1436,E2 835.9319} C_DIS
LIN {X 125.03,Y -58.3698,Z 163,A -27.9687,B 24.9656,C -1.355,E1 25.1452,E2 834.5989} C_DIS
LIN {X 127.8713,Y -51.8489,Z 163,A -24.5076,B 24.9636,C -1.394,E1 25.149,E2 831.0649} C_DIS
LIN {X 129.3913,Y -47.9316,Z 163,A -23.0825,B 24.9643,C -1.3808,E1 25.1504,E2 829.6788} C_DIS
LIN {X 130.8531,Y -43.7816,Z 163,A -21.4619,B 24.9646,C -1.3746,E1 25.1518,E2 828.0819} C_DIS
LIN {X 131.7834,Y -40.8994,Z 163,A -20.1599,B 24.9643,C -1.3812,E1 25.1529,E2 826.7717} C_DIS
LIN {X 132.7416,Y -37.6736,Z 163,A -18.7318,B 24.9639,C -1.3876,E1 25.1541,E2 825.3368} C_DIS
LIN {X 133.7461,Y -33.9311,Z 163,A -17.1497,B 24.9637,C -1.3913,E1 25.1552,E2 823.755} C_DIS
LIN {X 134.7884,Y -29.5231,Z 163,A -15.2887,B 24.9635,C -1.3963,E1 25.1563,E2 821.893} C_DIS
LIN {X 135.7058,Y -24.9756,Z 163,A -13.3041,B 24.963,C -1.4061,E1 25.1574,E2 819.8969} C_DIS
LIN {X 136.2816,Y -21.609,Z 163,A -11.2587,B 24.9607,C -1.4478,E1 25.1583,E2 817.7655} C_DIS
LIN {X 137.0521,Y -16.0074,Z 163,A -9.6966,B 24.9628,C -1.4093,E1 25.1588,E2 816.3032} C_DIS
LIN {X 137.456,Y -12.0611,Z 163,A -7.9397,B 24.9622,C -1.4212,E1 25.1593,E2 814.5286} C_DIS
LIN {X 137.7189,Y -8.5398,Z 163,A -5.9515,B 24.9602,C -1.4568,E1 25.1597,E2 812.4684} C_DIS
LIN {X 137.94,Y -3.482,Z 163,A -4.4739,B 24.9619,C -1.4271,E1 25.1597,E2 811.0696} C_DIS
LIN {X 137.9653,Y 2.2442,Z 163,A -2.0912,B 24.9614,C -1.4353,E1 25.1597,E2 808.6818} C_DIS
LIN {X 137.895,Y 4.9575,Z 163,A -0.2742,B 24.959,C -1.4795,E1 25.1596,E2 806.7713} C_DIS
LIN {X 137.5767,Y 10.6015,Z 163,A 1.5818,B 24.9602,C -1.4583,E1 25.1592,E2 804.9763} C_DIS
LIN {X 136.9472,Y 16.8864,Z 163,A 3.8466,B 24.9608,C -1.446,E1 25.1585,E2 802.7539} C_DIS
LIN {X 136.5925,Y 19.542,Z 163,A 5.4414,B 24.9591,C -1.4779,E1 25.1579,E2 801.0934} C_DIS
LIN {X 135.9716,Y 23.4886,Z 163,A 6.8248,B 24.9597,C -1.4671,E1 25.1572,E2 799.7436} C_DIS
LIN {X 135.2587,Y 27.2856,Z 163,A 8.2973,B 24.9598,C -1.4646,E1 25.1564,E2 798.2855} C_DIS
LIN {X 134.5795,Y 30.4595,Z 163,A 9.6304,B 24.9596,C -1.4681,E1 25.1556,E2 796.9521} C_DIS
LIN {X 133.7761,Y 33.8129,Z 163,A 11.0442,B 24.9594,C -1.4716,E1 25.1547,E2 795.5381} C_DIS
LIN {X 132.8462,Y 37.2994,Z 163,A 12.5527,B 24.9591,C -1.4769,E1 25.1536,E2 794.0257} C_DIS
LIN {X 132.0226,Y 40.1179,Z 163,A 14.2292,B 24.9574,C -1.5073,E1 25.1522,E2 792.2871} C_DIS
LIN {X 130.6683,Y 44.3366,Z 163,A 15.6482,B 24.9585,C -1.4884,E1 25.151,E2 790.9206} C_DIS
LIN {X 129.379,Y 47.9646,Z 163,A 17.212,B 24.9583,C -1.4913,E1 25.1495,E2 789.3588} C_DIS
LIN {X 128.016,Y 51.49,Z 163,A 18.6828,B 24.9583,C -1.4904,E1 25.148,E2 787.8984} C_DIS
LIN {X 126.6707,Y 54.7159,Z 163,A 20.1565,B 24.9581,C -1.496,E1 25.1464,E2 786.4195} C_DIS
LIN {X 125.3126,Y 57.7588,Z 163,A 21.5565,B 24.9578,C -1.501,E1 25.1447,E2 785.0153} C_DIS
LIN {X 123.8081,Y 60.9167,Z 163,A 22.9238,B 24.9578,C -1.5003,E1 25.1431,E2 783.6569} C_DIS
LIN {X 122.3433,Y 63.8086,Z 163,A 24.3677,B 24.9573,C -1.5098,E1 25.1412,E2 782.1983} C_DIS
LIN {X 120.1958,Y 67.7705,Z 163,A 26.2305,B 24.957,C -1.5145,E1 25.1387,E2 780.3341} C_DIS
LIN {X 118.0705,Y 71.4086,Z 163,A 28.007,B 24.9567,C -1.5209,E1 25.1362,E2 778.5516} C_DIS
LIN {X 115.7251,Y 75.1501,Z 163,A 29.846,B 24.9564,C -1.5262,E1 25.1334,E2 776.7096} C_DIS
LIN {X 112.526,Y 79.8617,Z 163,A 32.1481,B 24.9562,C -1.5287,E1 25.1297,E2 774.4127} C_DIS
LIN {X 110.0352,Y 83.2593,Z 163,A 33.9474,B 24.9558,C -1.5361,E1 25.1267,E2 772.6048} C_DIS
LIN {X 107.1616,Y 86.9273,Z 163,A 35.8824,B 24.9555,C -1.5408,E1 25.1234,E2 770.6674} C_DIS
LIN {X 104.3608,Y 90.2703,Z 163,A 37.4894,B 24.9559,C -1.5335,E1 25.1205,E2 769.085} C_DIS
LIN {X 99.5378,Y 95.5623,Z 163,A 40.7526,B 24.9546,C -1.5569,E1 25.1142,E2 765.7811} C_DIS
LIN {X 96.1356,Y 98.9839,Z 163,A 42.7087,B 24.9545,C -1.5586,E1 25.1103,E2 763.8292} C_DIS
LIN {X 92.3907,Y 102.4889,Z 163,A 44.7751,B 24.9545,C -1.5594,E1 25.1061,E2 761.7692} C_DIS
LIN {X 90.0717,Y 104.5319,Z 163,A 46.3639,B 24.9533,C -1.5794,E1 25.1027,E2 760.1394} C_DIS
LIN {X 86.8951,Y 107.1876,Z 163,A 47.705,B 24.9543,C -1.5612,E1 25.0999,E2 758.8463} C_DIS
LIN {X 83.7946,Y 109.628,Z 163,A 49.3567,B 24.9541,C -1.5651,E1 25.0962,E2 757.1916} C_DIS
LIN {X 80.3971,Y 112.1435,Z 163,A 50.9568,B 24.9544,C -1.5595,E1 25.0926,E2 755.6104} C_DIS
LIN {X 77.2701,Y 114.3205,Z 163,A 52.6867,B 24.9538,C -1.5705,E1 25.0886,E2 753.8604} C_DIS
LIN {X 73.4512,Y 116.811,Z 163,A 54.5762,B 24.9536,C -1.5734,E1 25.0842,E2 751.9702} C_DIS
LIN {X 69.6471,Y 119.1184,Z 163,A 56.4231,B 24.9535,C -1.5761,E1 25.0797,E2 750.1224} C_DIS
LIN {X 65.6683,Y 121.3577,Z 163,A 58.328,B 24.9533,C -1.5794,E1 25.0751,E2 748.2155} C_DIS
LIN {X 62.1255,Y 123.2071,Z 163,A 59.9988,B 24.9531,C -1.5822,E1 25.0709,E2 746.5424} C_DIS
LIN {X 58.3247,Y 125.0509,Z 163,A 61.5689,B 24.9536,C -1.5742,E1 25.067,E2 744.9955} C_DIS
LIN {X 55.0454,Y 126.5283,Z 163,A 63.2036,B 24.953,C -1.5838,E1 25.0628,E2 743.3421} C_DIS
LIN {X 51.953,Y 127.8293,Z 163,A 64.5983,B 24.953,C -1.5853,E1 25.0592,E2 741.9469} C_DIS
LIN {X 48.0512,Y 129.3466,Z 163,A 66.2532,B 24.953,C -1.5824,E1 25.0549,E2 740.3024} C_DIS
LIN {X 44.0417,Y 130.7665,Z 163,A 67.9917,B 24.953,C -1.5824,E1 25.0503,E2 738.5673} C_DIS
LIN {X 40.8731,Y 131.7914,Z 163,A 69.41,B 24.9529,C -1.5856,E1 25.0465,E2 737.1443} C_DIS
LIN {X 37.6495,Y 132.7483,Z 163,A 70.8118,B 24.9529,C -1.5869,E1 25.0428,E2 735.7418} C_DIS
LIN {X 34.0174,Y 133.7242,Z 163,A 72.3251,B 24.9529,C -1.5853,E1 25.0387,E2 734.2346} C_DIS
LIN {X 30.5628,Y 134.5559,Z 163,A 73.8233,B 24.9528,C -1.5873,E1 25.0346,E2 732.7337} C_DIS
LIN {X 26.4032,Y 135.4345,Z 163,A 75.6227,B 24.9526,C -1.59,E1 25.0297,E2 730.9301} C_DIS
LIN {X 18.5979,Y 136.7252,Z 163,A 79.0662,B 24.9521,C -1.5997,E1 25.0201,E2 727.467} C_DIS
LIN {X 12.266,Y 137.4384,Z 163,A 81.6732,B 24.9521,C -1.5979,E1 25.0129,E2 724.8659} C_DIS
LIN {X 8.9856,Y 137.6915,Z 163,A 83.3193,B 24.9512,C -1.6132,E1 25.0082,E2 723.1841} C_DIS
LIN {X 4.7525,Y 137.903,Z 163,A 84.7318,B 24.9524,C -1.5941,E1 25.0044,E2 721.8173} C_DIS
LIN {X -3.1647,Y 137.9485,Z 163,A 87.8742,B 24.9529,C -1.5856,E1 24.9957,E2 718.6954} C_DIS
LIN {X -9.4187,Y 137.663,Z 163,A 90.6161,B 24.9525,C -1.5923,E1 24.988,E2 715.9368} C_DIS
LIN {X -13.9125,Y 137.2815,Z 163,A 92.7594,B 24.9517,C -1.6059,E1 24.9819,E2 713.76} C_DIS
LIN {X -17.5596,Y 136.862,Z 163,A 94.3188,B 24.9517,C -1.6069,E1 24.9776,E2 712.1972} C_DIS
LIN {X -21.418,Y 136.3112,Z 163,A 95.6171,B 24.9527,C -1.5885,E1 24.9741,E2 710.9413} C_DIS
LIN {X -25.5778,Y 135.5923,Z 163,A 97.3157,B 24.953,C -1.5842,E1 24.9695,E2 709.2511} C_DIS
LIN {X -28.9582,Y 134.9104,Z 163,A 98.7684,B 24.953,C -1.5841,E1 24.9655,E2 707.797} C_DIS
LIN {X -32.4301,Y 134.118,Z 163,A 100.237,B 24.953,C -1.5822,E1 24.9615,E2 706.331} C_DIS
LIN {X -36.6255,Y 133.0347,Z 163,A 102.4385,B 24.9519,C -1.6017,E1 24.9555,E2 704.0797} C_DIS
LIN {X -40.4239,Y 131.9289,Z 163,A 103.6876,B 24.9533,C -1.5789,E1 24.9523,E2 702.8827} C_DIS
LIN {X -44.4735,Y 130.6217,Z 163,A 105.5454,B 24.9531,C -1.5814,E1 24.9473,E2 701.0154} C_DIS
LIN {X -47.7062,Y 129.4758,Z 163,A 107.1312,B 24.9527,C -1.5881,E1 24.9431,E2 699.4105} C_DIS
LIN {X -50.6994,Y 128.3333,Z 163,A 108.5164,B 24.9527,C -1.5892,E1 24.9395,E2 698.0198} C_DIS
LIN {X -53.9557,Y 126.9992,Z 163,A 109.7611,B 24.9535,C -1.5755,E1 24.9364,E2 696.8046} C_DIS
LIN {X -57.6017,Y 125.3852,Z 163,A 111.319,B 24.9539,C -1.5679,E1 24.9324,E2 695.2611} C_DIS
LIN {X -60.8022,Y 123.8646,Z 163,A 112.8468,B 24.9539,C -1.5685,E1 24.9286,E2 693.728} C_DIS
LIN {X -64.7514,Y 121.8482,Z 163,A 115.6561,B 24.951,C -1.6165,E1 24.9214,E2 690.7967} C_DIS
LIN {X -71.0579,Y 118.2825,Z 163,A 117.4942,B 24.955,C -1.5491,E1 24.9173,E2 689.1132} C_DIS
LIN {X -75.7358,Y 115.3428,Z 163,A 120.0731,B 24.9544,C -1.5595,E1 24.9112,E2 686.5015} C_DIS
LIN {X -79.3051,Y 112.9186,Z 163,A 121.8565,B 24.9547,C -1.5554,E1 24.9071,E2 684.7218} C_DIS
LIN {X -82.7816,Y 110.3957,Z 163,A 123.6476,B 24.9549,C -1.5519,E1 24.903,E2 682.9325} C_DIS
LIN {X -86.2927,Y 107.6735,Z 163,A 125.5503,B 24.9549,C -1.5509,E1 24.8989,E2 681.0253} C_DIS
LIN {X -89.6458,Y 104.898,Z 163,A 127.3279,B 24.9553,C -1.5452,E1 24.8951,E2 679.2544} C_DIS
LIN {X -92.856,Y 102.0667,Z 163,A 129.106,B 24.9555,C -1.541,E1 24.8914,E2 677.479} C_DIS
LIN {X -96.2012,Y 98.9205,Z 163,A 131.0415,B 24.9557,C -1.5379,E1 24.8875,E2 675.5431} C_DIS
LIN {X -99.4579,Y 95.6459,Z 163,A 132.9952,B 24.9559,C -1.5349,E1 24.8837,E2 673.5881} C_DIS
LIN {X -102.4537,Y 92.4296,Z 163,A 134.7918,B 24.9562,C -1.5287,E1 24.8803,E2 671.7983} C_DIS
LIN {X -105.0527,Y 89.4638,Z 163,A 136.7096,B 24.9556,C -1.5389,E1 24.8768,E2 669.8476} C_DIS
LIN {X -107.4191,Y 86.6081,Z 163,A 138.0857,B 24.9564,C -1.5262,E1 24.8744,E2 668.4951} C_DIS
LIN {X -110.3408,Y 82.8544,Z 163,A 139.9948,B 24.9569,C -1.5173,E1 24.8712,E2 666.5981} C_DIS
LIN {X -112.7643,Y 79.5239,Z 163,A 142.1558,B 24.9558,C -1.5358,E1 24.8676,E2 664.3826} C_DIS
LIN {X -115.4387,Y 75.5898,Z 163,A 143.5297,B 24.9579,C -1.4991,E1 24.8656,E2 663.0892} C_DIS
LIN {X -117.2254,Y 72.7877,Z 163,A 145.0858,B 24.9576,C -1.5041,E1 24.8633,E2 661.5132} C_DIS
LIN {X -119.6412,Y 68.746,Z 163,A 147.0779,B 24.9578,C -1.5002,E1 24.8604,E2 659.5202} C_DIS
LIN {X -121.9872,Y 64.4868,Z 163,A 148.9795,B 24.9585,C -1.4881,E1 24.8579,E2 657.6373} C_DIS
LIN {X -123.5875,Y 61.364,Z 163,A 150.5447,B 24.9585,C -1.4892,E1 24.856,E2 656.0611} C_DIS
LIN {X -125.164,Y 58.0801,Z 163,A 151.9571,B 24.959,C -1.4794,E1 24.8543,E2 654.6643} C_DIS
LIN {X -126.5877,Y 54.9078,Z 163,A 153.3896,B 24.9593,C -1.4743,E1 24.8527,E2 653.236} C_DIS
LIN {X -128.5029,Y 50.2631,Z 163,A 155.7777,B 24.9588,C -1.4832,E1 24.8502,E2 650.8135} C_DIS
LIN {X -130.2853,Y 45.4436,Z 163,A 157.6676,B 24.9599,C -1.4639,E1 24.8484,E2 648.9588} C_DIS
LIN {X -131.1987,Y 42.7416,Z 163,A 158.8302,B 24.9601,C -1.4589,E1 24.8474,E2 647.8014} C_DIS
LIN {X -132.2574,Y 39.3404,Z 163,A 160.4573,B 24.96,C -1.4617,E1 24.8461,E2 646.1584} C_DIS
LIN {X -133.3656,Y 35.3974,Z 163,A 162.1146,B 24.9604,C -1.4539,E1 24.8449,E2 644.5098} C_DIS
LIN {X -134.4262,Y 31.1309,Z 163,A 163.9085,B 24.9608,C -1.4463,E1 24.8437,E2 642.7236} C_DIS
LIN {X -135.1573,Y 27.7841,Z 163,A 165.3635,B 24.961,C -1.4433,E1 24.8429,E2 641.2672} C_DIS
LIN {X -135.8231,Y 24.3197,Z 163,A 166.8451,B 24.9612,C -1.4393,E1 24.8421,E2 639.7863} C_DIS
LIN {X -136.5152,Y 20.0824,Z 163,A 168.6675,B 24.9614,C -1.4354,E1 24.8413,E2 637.9623} C_DIS
LIN {X -137.0226,Y 16.2544,Z 163,A 170.2088,B 24.9619,C -1.427,E1 24.8408,E2 636.4321} C_DIS
LIN {X -137.4182,Y 12.4955,Z 163,A 171.8881,B 24.9619,C -1.4273,E1 24.8403,E2 634.7419} C_DIS
LIN {X -137.6949,Y 8.9289,Z 163,A 173.1855,B 24.9626,C -1.4128,E1 24.8401,E2 633.4712} C_DIS
LIN {X -137.8795,Y 5.3547,Z 163,A 174.8358,B 24.9624,C -1.4162,E1 24.8399,E2 631.8028} C_DIS
LIN {X -137.9815,Y 0.8871,Z 163,A 176.6486,B 24.9629,C -1.4079,E1 24.8398,E2 629.999} C_DIS
LIN {X -137.9528,Y -2.9915,Z 163,A 178.3836,B 24.9629,C -1.4089,E1 24.8398,E2 628.2512} C_DIS
LIN {X -137.8202,Y -6.7132,Z 163,A 179.8581,B 24.9633,C -1.4001,E1 24.84,E2 626.7887} C_DIS
LIN {X -137.6018,Y -10.2573,Z 163,A -178.6578,B 24.9635,C -1.3957,E1 24.8403,E2 625.3061} C_DIS
LIN {X -137.2176,Y -14.5191,Z 163,A -176.862,B 24.9638,C -1.3909,E1 24.8408,E2 623.5111} C_DIS
LIN {X -136.7687,Y -18.2713,Z 163,A -175.2118,B 24.9638,C -1.3899,E1 24.8414,E2 621.8534} C_DIS
LIN {X -136.1393,Y -22.4835,Z 163,A -173.5579,B 24.9644,C -1.3783,E1 24.8421,E2 620.2174} C_DIS
LIN {X -135.5437,Y -25.8318,Z 163,A -172.1374,B 24.9646,C -1.3741,E1 24.8428,E2 618.7983} C_DIS
LIN {X -134.9306,Y -28.8644,Z 163,A -170.8003,B 24.9647,C -1.3727,E1 24.8436,E2 617.4566} C_DIS
LIN {X -134.1708,Y -32.2114,Z 163,A -169.4229,B 24.9651,C -1.3657,E1 24.8445,E2 616.0878} C_DIS
LIN {X -133.3897,Y -35.3073,Z 163,A -168.2316,B 24.9656,C -1.3547,E1 24.8453,E2 614.9159} C_DIS
LIN {X -131.6957,Y -41.1853,Z 163,A -165.502,B 24.9656,C -1.3563,E1 24.8474,E2 612.1667} C_DIS
LIN {X -130.2718,Y -45.4826,Z 163,A -163.6002,B 24.9658,C -1.3517,E1 24.8491,E2 610.265} C_DIS
LIN {X -129.2453,Y -48.3215,Z 163,A -162.2139,B 24.9656,C -1.3547,E1 24.8505,E2 608.8636} C_DIS
LIN {X -127.4722,Y -52.823,Z 163,A -160.2731,B 24.9661,C -1.3452,E1 24.8525,E2 606.9348} C_DIS
LIN {X -126.0359,Y -56.1629,Z 163,A -158.1069,B 24.9646,C -1.3748,E1 24.8551,E2 604.686} C_DIS
LIN {X -123.7279,Y -61.0794,Z 163,A -156.6481,B 24.967,C -1.3269,E1 24.8567,E2 603.3335} C_DIS
LIN {X -122.3094,Y -63.8732,Z 163,A -155.2456,B 24.967,C -1.3284,E1 24.8585,E2 601.9198} C_DIS
LIN {X -120.7168,Y -66.8378,Z 163,A -153.6635,B 24.9667,C -1.334,E1 24.8607,E2 600.3161} C_DIS
LIN {X -118.3711,Y -70.9099,Z 163,A -151.7597,B 24.9671,C -1.3262,E1 24.8633,E2 598.4211} C_DIS
LIN {X -116.0081,Y -74.7135,Z 163,A -150.0675,B 24.9677,C -1.3125,E1 24.8658,E2 596.7529} C_DIS
LIN {X -111.4253,Y -81.3902,Z 163,A -146.2174,B 24.9669,C -1.3291,E1 24.8721,E2 592.8442} C_DIS
LIN {X -109.1771,Y -84.3814,Z 163,A -144.96,B 24.9679,C -1.3097,E1 24.8742,E2 591.6271} C_DIS
LIN {X -106.5141,Y -87.7195,Z 163,A -143.2074,B 24.9681,C -1.3043,E1 24.8772,E2 589.8792} C_DIS
LIN {X -103.919,Y -90.7774,Z 163,A -141.2,B 24.9674,C -1.3184,E1 24.881,E2 587.8292} C_DIS
LIN {X -101.3578,Y -93.6298,Z 163,A -139.8871,B 24.9683,C -1.3,E1 24.8834,E2 586.5542} C_DIS
LIN {X -98.2392,Y -96.897,Z 163,A -137.9845,B 24.9685,C -1.2972,E1 24.8871,E2 584.65} C_DIS
LIN {X -95.2142,Y -99.8704,Z 163,A -136.2526,B 24.9687,C -1.2919,E1 24.8906,E2 582.9235} C_DIS
LIN {X -92.2237,Y -102.6385,Z 163,A -133.8618,B 24.9671,C -1.3256,E1 24.8957,E2 580.4432} C_DIS
LIN {X -87.7781,Y -106.4656,Z 163,A -132.0754,B 24.969,C -1.2862,E1 24.8994,E2 578.7436} C_DIS
LIN {X -84.222,Y -109.3007,Z 163,A -130.3416,B 24.9696,C -1.2744,E1 24.9031,E2 577.0313} C_DIS
LIN {X -80.73,Y -111.9044,Z 163,A -128.3671,B 24.9693,C -1.28,E1 24.9076,E2 575.0367} C_DIS
LIN {X -77.0396,Y -114.4765,Z 163,A -126.4874,B 24.9694,C -1.2775,E1 24.9119,E2 573.1566} C_DIS
LIN {X -73.3613,Y -116.8677,Z 163,A -124.6741,B 24.9696,C -1.2741,E1 24.9162,E2 571.3454} C_DIS
LIN {X -69.5644,Y -119.167,Z 163,A -122.8081,B 24.9696,C -1.2726,E1 24.9207,E2 569.4775} C_DIS
LIN {X -65.6406,Y -121.3725,Z 163,A -120.9057,B 24.9697,C -1.2717,E1 24.9254,E2 567.5716} C_DIS
LIN {X -61.4836,Y -123.5285,Z 163,A -119.0652,B 24.9701,C -1.2636,E1 24.9299,E2 565.7454} C_DIS
LIN {X -58.1868,Y -125.1147,Z 163,A -117.4348,B 24.9699,C -1.2678,E1 24.9341,E2 564.101} C_DIS
LIN {X -54.3954,Y -126.8093,Z 163,A -115.7043,B 24.9699,C -1.2662,E1 24.9385,E2 562.3702} C_DIS
LIN {X -50.2954,Y -128.4904,Z 163,A -113.9396,B 24.9703,C -1.2602,E1 24.943,E2 560.6157} C_DIS
LIN {X -46.1949,Y -130.0221,Z 163,A -112.0939,B 24.9703,C -1.2601,E1 24.9479,E2 558.7667} C_DIS
LIN {X -42.2498,Y -131.3558,Z 163,A -110.4452,B 24.9705,C -1.2543,E1 24.9522,E2 557.1287} C_DIS
LIN {X -39.0333,Y -132.3473,Z 163,A -109.0398,B 24.9705,C -1.2537,E1 24.956,E2 555.7224} C_DIS
LIN {X -35.7344,Y -133.2758,Z 163,A -107.6643,B 24.9707,C -1.2502,E1 24.9597,E2 554.3531} C_DIS
LIN {X -32.403,Y -134.1246,Z 163,A -106.193,B 24.9707,C -1.2517,E1 24.9637,E2 552.8759} C_DIS
LIN {X -29.762,Y -134.7368,Z 163,A -104.8984,B 24.9702,C -1.2604,E1 24.9673,E2 551.5593} C_DIS
LIN {X -21.1759,Y -136.3487,Z 163,A -101.4343,B 24.9707,C -1.2501,E1 24.9767,E2 548.116} C_DIS
LIN {X -18.5465,Y -136.7326,Z 163,A -99.7913,B 24.9693,C -1.2795,E1 24.9815,E2 546.4019} C_DIS
LIN {X -13.9761,Y -137.2746,Z 163,A -98.1772,B 24.9701,C -1.2629,E1 24.9859,E2 544.8265} C_DIS
LIN {X -8.6695,Y -137.7109,Z 163,A -96.1604,B 24.9706,C -1.2521,E1 24.9914,E2 542.8343} C_DIS
LIN {X -4.8727,Y -137.8983,Z 163,A -94.2453,B 24.9697,C -1.2709,E1 24.9969,E2 540.8743} C_DIS
LIN {X -1.1149,Y -137.9795,Z 163,A -92.7526,B 24.9699,C -1.2675,E1 25.001,E2 539.3897} C_DIS
LIN {X -1.1149,Y -137.9795,Z 163,A -92.7526,B 24.9699,C -1.2675,E1 25.001,E2 539.3897} C_DIS
Enddeposition()
LIN {X 0.9656,Y -137.0582,Z 163,A -91.525,B 22.0645,C -0.7344,E1 22.0778,E2 539.1567} C_DIS
Startdeposition()
$VEL.CP = VEL_PRINT
LIN {X -5.51,Y -136.9519,Z 163,A -94.542,B 22.065,C -0.7191,E1 22.0692,E2 542.2147} C_DIS
LIN {X -12.1846,Y -136.5214,Z 163,A -97.2115,B 22.0648,C -0.7251,E1 22.0618,E2 544.8694} C_DIS
LIN {X -18.0222,Y -135.8725,Z 163,A -99.8566,B 22.0651,C -0.7165,E1 22.0544,E2 547.5394} C_DIS
LIN {X -20.6362,Y -135.5004,Z 163,A -102.189,B 22.0668,C -0.6595,E1 22.0476,E2 550.0259} C_DIS
LIN {X -28.9687,Y -133.966,Z 163,A -104.4566,B 22.065,C -0.7202,E1 22.0418,E2 552.1347} C_DIS
LIN {X -32.0483,Y -133.2628,Z 163,A -105.803,B 22.065,C -0.7197,E1 22.0381,E2 553.4845} C_DIS
LIN {X -35.4694,Y -132.3933,Z 163,A -107.2949,B 22.065,C -0.7199,E1 22.0341,E2 554.9786} C_DIS
LIN {X -39.5175,Y -131.2432,Z 163,A -109.1433,B 22.065,C -0.7169,E1 22.0291,E2 556.8383} C_DIS
LIN {X -43.3465,Y -130.0274,Z 163,A -110.7032,B 22.0649,C -0.7238,E1 22.025,E2 558.3831} C_DIS
LIN {X -46.1998,Y -129.0414,Z 163,A -111.9611,B 22.0649,C -0.7251,E1 22.0217,E2 559.6403} C_DIS
LIN {X -49.3885,Y -127.8549,Z 163,A -113.3808,B 22.0648,C -0.7266,E1 22.018,E2 561.0596} C_DIS
LIN {X -52.2093,Y -126.7306,Z 163,A -115.086,B 22.0654,C -0.7078,E1 22.0134,E2 562.8194} C_DIS
LIN {X -55.6943,Y -125.2367,Z 163,A -116.1584,B 22.0646,C -0.7332,E1 22.0109,E2 563.8269} C_DIS
LIN {X -59.5955,Y -123.4289,Z 163,A -118.1614,B 22.0648,C -0.7258,E1 22.0057,E2 565.8554} C_DIS
LIN {X -63.2911,Y -121.5749,Z 163,A -119.8464,B 22.0647,C -0.73,E1 22.0015,E2 567.5344} C_DIS
LIN {X -67.0688,Y -119.5338,Z 163,A -121.7158,B 22.0647,C -0.729,E1 21.9969,E2 569.4126} C_DIS
LIN {X -71.1851,Y -117.1294,Z 163,A -123.7054,B 22.0647,C -0.7321,E1 21.9922,E2 571.4008} C_DIS
LIN {X -75.005,Y -114.7213,Z 163,A -125.6293,B 22.0646,C -0.7334,E1 21.9876,E2 573.3284} C_DIS
LIN {X -78.7701,Y -112.169,Z 163,A -127.5185,B 22.0645,C -0.7371,E1 21.9833,E2 575.215} C_DIS
LIN {X -81.2863,Y -110.359,Z 163,A -129.1459,B 22.0649,C -0.7244,E1 21.9796,E2 576.8831} C_DIS
LIN {X -84.505,Y -107.9142,Z 163,A -130.2716,B 22.0639,C -0.7529,E1 21.9772,E2 577.9372} C_DIS
LIN {X -91.6611,Y -101.9062,Z 163,A -134.3602,B 22.0639,C -0.7521,E1 21.9685,E2 582.0462} C_DIS
LIN {X -94.7414,Y -99.0485,Z 163,A -136.1565,B 22.0639,C -0.7539,E1 21.9648,E2 583.8461} C_DIS
LIN {X -97.789,Y -96.0409,Z 163,A -137.9977,B 22.0639,C -0.7554,E1 21.9612,E2 585.6922} C_DIS
LIN {X -100.9439,Y -92.7192,Z 163,A -139.8325,B 22.0636,C -0.7633,E1 21.9577,E2 587.5152} C_DIS
LIN {X -104.7991,Y -88.339,Z 163,A -142.39,B 22.0636,C -0.7636,E1 21.953,E2 590.0853} C_DIS
LIN {X -107.4971,Y -85.0358,Z 163,A -144.0693,B 22.0633,C -0.7725,E1 21.9501,E2 591.7499} C_DIS
LIN {X -110.0223,Y -81.7413,Z 163,A -145.8792,B 22.0633,C -0.7734,E1 21.947,E2 593.5672} C_DIS
LIN {X -111.7673,Y -79.3397,Z 163,A -147.6793,B 22.064,C -0.7517,E1 21.944,E2 595.4355} C_DIS
LIN {X -114.5802,Y -75.2193,Z 163,A -149.2573,B 22.0631,C -0.7795,E1 21.9417,E2 596.9482} C_DIS
LIN {X -116.9667,Y -71.452,Z 163,A -151.1106,B 22.0629,C -0.7849,E1 21.9389,E2 598.7979} C_DIS
LIN {X -119.2322,Y -67.6043,Z 163,A -153.0042,B 22.0628,C -0.7887,E1 21.9363,E2 600.6927} C_DIS
LIN {X -121.19,Y -64.0241,Z 163,A -154.4392,B 22.0622,C -0.8054,E1 21.9344,E2 602.0917} C_DIS
LIN {X -123.4032,Y -59.6478,Z 163,A -157.2709,B 22.0632,C -0.7767,E1 21.9308,E2 605.0177} C_DIS
LIN {X -125.4503,Y -55.2168,Z 163,A -158.8326,B 22.0623,C -0.8035,E1 21.9291,E2 606.5177} C_DIS
LIN {X -127.0607,Y -51.3966,Z 163,A -160.5027,B 22.062,C -0.8113,E1 21.9273,E2 608.1774} C_DIS
LIN {X -128.62,Y -47.3656,Z 163,A -162.4302,B 22.062,C -0.8113,E1 21.9254,E2 610.1175} C_DIS
LIN {X -129.9335,Y -43.6284,Z 163,A -164.0034,B 22.0617,C -0.8199,E1 21.924,E2 611.6779} C_DIS
LIN {X -130.888,Y -40.6783,Z 163,A -165.4461,B 22.0617,C -0.8173,E1 21.9228,E2 613.137} C_DIS
LIN {X -132.4111,Y -35.403,Z 163,A -167.6116,B 22.0613,C -0.83,E1 21.9212,E2 615.2829} C_DIS
LIN {X -133.2334,Y -32.1704,Z 163,A -169.0117,B 22.0612,C -0.8341,E1 21.9202,E2 616.6816} C_DIS
LIN {X -134.0053,Y -28.7865,Z 163,A -170.4871,B 22.0611,C -0.8375,E1 21.9193,E2 618.1579} C_DIS
LIN {X -134.8464,Y -24.5498,Z 163,A -172.3253,B 22.0609,C -0.8417,E1 21.9184,E2 619.9972} C_DIS
LIN {X -135.4481,Y -20.9739,Z 163,A -173.7822,B 22.0606,C -0.8491,E1 21.9177,E2 621.4444} C_DIS
LIN {X -135.9098,Y -17.7379,Z 163,A -175.1974,B 22.0606,C -0.8513,E1 21.9172,E2 622.8635} C_DIS
LIN {X -136.3742,Y -13.7331,Z 163,A -176.9552,B 22.0605,C -0.8534,E1 21.9166,E2 624.6275} C_DIS
LIN {X -136.6899,Y -10.1002,Z 163,A -178.467,B 22.0603,C -0.8589,E1 21.9163,E2 626.1353} C_DIS
LIN {X -136.942,Y -5.7615,Z 163,A 179.7002,B 22.0601,C -0.864,E1 21.916,E2 627.967} C_DIS
LIN {X -137.051,Y -1.8333,Z 163,A 178.0927,B 22.0598,C -0.8708,E1 21.916,E2 629.5675} C_DIS
LIN {X -137.0437,Y 2.2767,Z 163,A 176.4296,B 22.0595,C -0.8787,E1 21.916,E2 631.2208} C_DIS
LIN {X -136.9292,Y 6.0824,Z 163,A 174.5255,B 22.0598,C -0.8702,E1 21.9162,E2 633.1608} C_DIS
LIN {X -136.5982,Y 11.2743,Z 163,A 172.5459,B 22.0593,C -0.8857,E1 21.9166,E2 635.1126} C_DIS
LIN {X -136.279,Y 14.6335,Z 163,A 171.1265,B 22.0591,C -0.8899,E1 21.917,E2 636.5306} C_DIS
LIN {X -135.7939,Y 18.6205,Z 163,A 169.3732,B 22.0591,C -0.892,E1 21.9176,E2 638.2903} C_DIS
LIN {X -135.262,Y 22.1462,Z 163,A 167.9134,B 22.0588,C -0.8982,E1 21.9182,E2 639.7435} C_DIS
LIN {X -134.6418,Y 25.6453,Z 163,A 166.4489,B 22.0586,C -0.9038,E1 21.919,E2 641.2029} C_DIS
LIN {X -133.9188,Y 29.1874,Z 163,A 164.896,B 22.0584,C -0.9068,E1 21.9199,E2 642.7583} C_DIS
LIN {X -132.9662,Y 33.2605,Z 163,A 163.1838,B 22.0582,C -0.914,E1 21.921,E2 644.463} C_DIS
LIN {X -132.1242,Y 36.4618,Z 163,A 161.7453,B 22.0581,C -0.9159,E1 21.922,E2 645.9057} C_DIS
LIN {X -130.9689,Y 40.414,Z 163,A 160.0026,B 22.0579,C -0.9204,E1 21.9234,E2 647.648} C_DIS
LIN {X -129.6315,Y 44.518,Z 163,A 158.222,B 22.0577,C -0.927,E1 21.925,E2 649.4225} C_DIS
LIN {X -128.4981,Y 47.691,Z 163,A 156.8407,B 22.0574,C -0.9326,E1 21.9263,E2 650.798} C_DIS
LIN {X -126.2674,Y 53.3182,Z 163,A 154.1578,B 22.0574,C -0.9336,E1 21.9291,E2 653.4953} C_DIS
LIN {X -124.5716,Y 57.167,Z 163,A 152.4775,B 22.057,C -0.9423,E1 21.931,E2 655.1629} C_DIS
LIN {X -123.4006,Y 59.6548,Z 163,A 151.1366,B 22.0572,C -0.9374,E1 21.9327,E2 656.5255} C_DIS
LIN {X -121.4995,Y 63.4347,Z 163,A 149.7434,B 22.0564,C -0.959,E1 21.9344,E2 657.8692} C_DIS
LIN {X -118.7907,Y 68.377,Z 163,A 147.0602,B 22.0567,C -0.9514,E1 21.9381,E2 660.5889} C_DIS
LIN {X -116.5126,Y 72.1902,Z 163,A 145.3871,B 22.0561,C -0.9648,E1 21.9404,E2 662.2363} C_DIS
LIN {X -114.8504,Y 74.8061,Z 163,A 144.1158,B 22.0559,C -0.9695,E1 21.9424,E2 663.5024} C_DIS
LIN {X -111.6194,Y 79.5468,Z 163,A 141.4703,B 22.0561,C -0.9652,E1 21.9466,E2 666.1744} C_DIS
LIN {X -109.7435,Y 82.1157,Z 163,A 140.0426,B 22.0561,C -0.9644,E1 21.949,E2 667.612} C_DIS
LIN {X -107.5548,Y 84.9623,Z 163,A 138.6026,B 22.0559,C -0.9711,E1 21.9515,E2 669.042} C_DIS
LIN {X -104.874,Y 88.2497,Z 163,A 136.8373,B 22.0556,C -0.976,E1 21.9546,E2 670.8035} C_DIS
LIN {X -101.8923,Y 91.6766,Z 163,A 134.9352,B 22.0554,C -0.9807,E1 21.9581,E2 672.703} C_DIS
LIN {X -98.8276,Y 94.9725,Z 163,A 133.0586,B 22.0552,C -0.9855,E1 21.9617,E2 674.5761} C_DIS
LIN {X -95.7044,Y 98.119,Z 163,A 131.244,B 22.055,C -0.9916,E1 21.9653,E2 676.3831} C_DIS
LIN {X -92.5871,Y 101.0654,Z 163,A 129.381,B 22.055,C -0.9927,E1 21.9691,E2 678.2519} C_DIS
LIN {X -89.1398,Y 104.1192,Z 163,A 127.4307,B 22.0548,C -0.9959,E1 21.9732,E2 680.2025} C_DIS
LIN {X -85.7208,Y 106.9516,Z 163,A 125.5545,B 22.0547,C -0.999,E1 21.9773,E2 682.0785} C_DIS
LIN {X -82.2506,Y 109.6427,Z 163,A 123.7545,B 22.0544,C -1.0044,E1 21.9812,E2 683.8715} C_DIS
LIN {X -78.7293,Y 112.1978,Z 163,A 122.019,B 22.0541,C -1.0118,E1 21.9852,E2 685.5942} C_DIS
LIN {X -76.1152,Y 113.9869,Z 163,A 120.5699,B 22.0542,C -1.0088,E1 21.9885,E2 687.0569} C_DIS
LIN {X -72.1434,Y 116.5417,Z 163,A 118.6114,B 22.0541,C -1.0132,E1 21.9932,E2 689.0108} C_DIS
LIN {X -69.216,Y 118.3036,Z 163,A 116.2867,B 22.0556,C -0.9759,E1 21.9991,E2 691.4431} C_DIS
LIN {X -63.1879,Y 121.6291,Z 163,A 114.3018,B 22.0537,C -1.0203,E1 22.0037,E2 693.3157} C_DIS
LIN {X -59.3616,Y 123.5406,Z 163,A 112.5607,B 22.0535,C -1.0253,E1 22.008,E2 695.0488} C_DIS
LIN {X -56.3467,Y 124.9449,Z 163,A 111.2266,B 22.0533,C -1.0299,E1 22.0114,E2 696.3744} C_DIS
LIN {X -53.2662,Y 126.2891,Z 163,A 109.9101,B 22.053,C -1.0359,E1 22.0147,E2 697.6783} C_DIS
LIN {X -47.5968,Y 128.5334,Z 163,A 107.3242,B 22.053,C -1.0375,E1 22.0214,E2 700.2662} C_DIS
LIN {X -42.9104,Y 130.1725,Z 163,A 105.2246,B 22.053,C -1.0389,E1 22.027,E2 702.3667} C_DIS
LIN {X -37.9137,Y 131.7155,Z 163,A 102.8076,B 22.0533,C -1.0308,E1 22.0335,E2 704.8102} C_DIS
LIN {X -34.067,Y 132.7615,Z 163,A 101.2466,B 22.053,C -1.0372,E1 22.0377,E2 706.3567} C_DIS
LIN {X -30.656,Y 133.59,Z 163,A 99.8003,B 22.0529,C -1.0395,E1 22.0416,E2 707.7991} C_DIS
LIN {X -27.361,Y 134.3036,Z 163,A 98.4839,B 22.0526,C -1.045,E1 22.0452,E2 709.1028} C_DIS
LIN {X -24.2509,Y 134.8999,Z 163,A 97.0097,B 22.0529,C -1.039,E1 22.0493,E2 710.5945} C_DIS
LIN {X -20.1206,Y 135.5795,Z 163,A 95.3525,B 22.0527,C -1.0444,E1 22.0538,E2 712.239} C_DIS
LIN {X -16.7896,Y 136.0313,Z 163,A 93.3469,B 22.0539,C -1.0177,E1 22.0596,E2 714.3175} C_DIS
LIN {X -12.1158,Y 136.5272,Z 163,A 91.8833,B 22.0528,C -1.0416,E1 22.0635,E2 715.7183} C_DIS
LIN {X -9.0898,Y 136.7624,Z 163,A 90.0039,B 22.054,C -1.014,E1 22.0689,E2 717.6721} C_DIS
LIN {X -3.9129,Y 137.0067,Z 163,A 87.767,B 22.0541,C -1.0113,E1 22.0752,E2 719.9163} C_DIS
LIN {X 1.7646,Y 137.0522,Z 163,A 86.0471,B 22.0528,C -1.0418,E1 22.0797,E2 721.5548} C_DIS
LIN {X 9.7922,Y 136.7124,Z 163,A 82.2374,B 22.0537,C -1.0209,E1 22.0905,E2 725.4187} C_DIS
LIN {X 14.3272,Y 136.312,Z 163,A 80.8232,B 22.0527,C -1.0434,E1 22.0943,E2 726.772} C_DIS
LIN {X 17.9677,Y 135.8797,Z 163,A 79.5389,B 22.0522,C -1.0547,E1 22.0977,E2 728.025} C_DIS
LIN {X 25.7519,Y 134.6214,Z 163,A 76.0258,B 22.0527,C -1.0432,E1 22.1075,E2 731.5646} C_DIS
LIN {X 29.3064,Y 133.8931,Z 163,A 74.4106,B 22.053,C -1.0378,E1 22.1119,E2 733.1918} C_DIS
LIN {X 33.3396,Y 132.9461,Z 163,A 72.763,B 22.0528,C -1.0407,E1 22.1164,E2 734.8288} C_DIS
LIN {X 36.7484,Y 132.044,Z 163,A 71.3445,B 22.0528,C -1.0424,E1 22.1202,E2 736.2403} C_DIS
LIN {X 39.964,Y 131.1066,Z 163,A 69.9603,B 22.0528,C -1.0421,E1 22.1239,E2 737.6226} C_DIS
LIN {X 43.1777,Y 130.0836,Z 163,A 68.4885,B 22.053,C -1.038,E1 22.1278,E2 739.1021} C_DIS
LIN {X 46.2748,Y 129.0144,Z 163,A 67.1456,B 22.053,C -1.038,E1 22.1313,E2 740.4418} C_DIS
LIN {X 49.666,Y 127.747,Z 163,A 65.343,B 22.0536,C -1.0227,E1 22.1361,E2 742.2805} C_DIS
LIN {X 52.7277,Y 126.5141,Z 163,A 64.4048,B 22.0528,C -1.0423,E1 22.1384,E2 743.164} C_DIS
LIN {X 56.6338,Y 124.8165,Z 163,A 62.3879,B 22.0534,C -1.0289,E1 22.1436,E2 745.211} C_DIS
LIN {X 60.184,Y 123.1427,Z 163,A 60.7718,B 22.0534,C -1.0281,E1 22.1477,E2 746.8244} C_DIS
LIN {X 63.5966,Y 121.4145,Z 163,A 59.2991,B 22.0532,C -1.0321,E1 22.1513,E2 748.2819} C_DIS
LIN {X 67.2024,Y 119.4587,Z 163,A 57.4516,B 22.0536,C -1.0232,E1 22.1559,E2 750.1467} C_DIS
LIN {X 71.1952,Y 117.1233,Z 163,A 55.5178,B 22.0537,C -1.0203,E1 22.1605,E2 752.0814} C_DIS
LIN {X 75.0042,Y 114.7218,Z 163,A 53.6162,B 22.0539,C -1.0163,E1 22.165,E2 753.9864} C_DIS
LIN {X 78.701,Y 112.2177,Z 163,A 51.7512,B 22.054,C -1.0133,E1 22.1693,E2 755.8522} C_DIS
LIN {X 82.2922,Y 109.6113,Z 163,A 49.9118,B 22.0542,C -1.0107,E1 22.1734,E2 757.6907} C_DIS
LIN {X 87.5662,Y 105.4444,Z 163,A 47.0438,B 22.0545,C -1.0026,E1 22.1797,E2 760.5679} C_DIS
LIN {X 91.532,Y 102.0218,Z 163,A 44.9708,B 22.0545,C -1.0039,E1 22.184,E2 762.6279} C_DIS
LIN {X 93.9449,Y 99.8044,Z 163,A 43.5095,B 22.0548,C -0.9966,E1 22.187,E2 764.1018} C_DIS
LIN {X 97.556,Y 96.2785,Z 163,A 41.4913,B 22.0548,C -0.9966,E1 22.191,E2 766.1103} C_DIS
LIN {X 102.9909,Y 90.4411,Z 163,A 38.1456,B 22.0551,C -0.9884,E1 22.1973,E2 769.4605} C_DIS
LIN {X 105.89,Y 87.0287,Z 163,A 36.3414,B 22.0551,C -0.9874,E1 22.2005,E2 771.258} C_DIS
LIN {X 108.6824,Y 83.5151,Z 163,A 34.4399,B 22.0554,C -0.9816,E1 22.2038,E2 773.1646} C_DIS
LIN {X 110.5278,Y 81.0564,Z 163,A 33.0365,B 22.0558,C -0.9725,E1 22.2062,E2 774.5843} C_DIS
LIN {X 113.7979,Y 76.3983,Z 163,A 30.7782,B 22.0558,C -0.9725,E1 22.2097,E2 776.83} C_DIS
LIN {X 116.3137,Y 72.5097,Z 163,A 28.8979,B 22.0558,C -0.9701,E1 22.2125,E2 778.7055} C_DIS
LIN {X 118.5174,Y 68.8492,Z 163,A 27.0996,B 22.0561,C -0.9647,E1 22.2151,E2 780.5075} C_DIS
LIN {X 120.8265,Y 64.7111,Z 163,A 25.0764,B 22.0564,C -0.9572,E1 22.2178,E2 782.5386} C_DIS
LIN {X 122.6866,Y 61.1087,Z 163,A 23.4816,B 22.0564,C -0.9574,E1 22.2198,E2 784.1228} C_DIS
LIN {X 124.2992,Y 57.756,Z 163,A 21.9883,B 22.0564,C -0.9561,E1 22.2216,E2 785.6103} C_DIS
LIN {X 125.6887,Y 54.6666,Z 163,A 20.5909,B 22.0566,C -0.953,E1 22.2231,E2 787.0072} C_DIS
LIN {X 126.9086,Y 51.7741,Z 163,A 19.2513,B 22.0568,C -0.9478,E1 22.2246,E2 788.3521} C_DIS
LIN {X 128.2647,Y 48.3141,Z 163,A 17.7501,B 22.0568,C -0.9459,E1 22.2261,E2 789.8489} C_DIS
LIN {X 130.5191,Y 41.8427,Z 163,A 14.7375,B 22.0575,C -0.9298,E1 22.2288,E2 792.8843} C_DIS
LIN {X 131.8896,Y 37.3005,Z 163,A 12.9092,B 22.0575,C -0.9316,E1 22.2302,E2 794.696} C_DIS
LIN {X 132.8057,Y 33.8929,Z 163,A 11.5049,B 22.0575,C -0.9307,E1 22.2312,E2 796.0936} C_DIS
LIN {X 133.6014,Y 30.6061,Z 163,A 10.0702,B 22.0577,C -0.9252,E1 22.2321,E2 797.5331} C_DIS
LIN {X 134.3646,Y 27.0609,Z 163,A 8.5529,B 22.0579,C -0.9204,E1 22.233,E2 799.0529} C_DIS
LIN {X 135.1455,Y 22.8446,Z 163,A 7.0052,B 22.0576,C -0.9272,E1 22.2338,E2 800.5723} C_DIS
LIN {X 135.8755,Y 17.9997,Z 163,A 4.7553,B 22.0583,C -0.9104,E1 22.2347,E2 802.8512} C_DIS
LIN {X 136.3037,Y 14.4039,Z 163,A 3.4121,B 22.0582,C -0.9143,E1 22.2351,E2 804.1751} C_DIS
LIN {X 136.5534,Y 11.8054,Z 163,A 2.1255,B 22.0587,C -0.9009,E1 22.2354,E2 805.4885} C_DIS
LIN {X 136.9879,Y 4.5857,Z 163,A -0.8078,B 22.0589,C -0.8957,E1 22.2359,E2 808.4154} C_DIS
LIN {X 137.0637,Y 0.4089,Z 163,A -2.8012,B 22.0596,C -0.8776,E1 22.2359,E2 810.4432} C_DIS
LIN {X 136.9336,Y -5.9766,Z 163,A -5.1722,B 22.0593,C -0.8841,E1 22.2358,E2 812.7807} C_DIS
LIN {X 136.7208,Y -9.6772,Z 163,A -6.5398,B 22.0592,C -0.8884,E1 22.2355,E2 814.1277} C_DIS
LIN {X 135.9689,Y -17.2869,Z 163,A -10.3661,B 22.0607,C -0.8461,E1 22.2344,E2 818.0399} C_DIS
LIN {X 135.3858,Y -21.3765,Z 163,A -11.7007,B 22.0602,C -0.8603,E1 22.2338,E2 819.3277} C_DIS
LIN {X 134.6721,Y -25.4867,Z 163,A -13.3619,B 22.0602,C -0.8589,E1 22.233,E2 820.9814} C_DIS
LIN {X 133.823,Y -29.6293,Z 163,A -15.5551,B 22.0613,C -0.8317,E1 22.2317,E2 823.2319} C_DIS
LIN {X 132.9,Y -33.5215,Z 163,A -16.7154,B 22.0605,C -0.8524,E1 22.2309,E2 824.33} C_DIS
Enddeposition()
END
